LIN {X 0,Y 453.456,Z 225.499,A -85,B 0,C 180,E1 -8413.244,E2 -8413.244} C_VEL
LIN {X 0,Y 453.465,Z 225.498,A -85,B 0,C 180,E1 -8415.778,E2 -8415.778} C_VEL
LIN {X 0,Y 453.48,Z 225.494,A -85,B 0,C 180,E1 -8418.209,E2 -8418.209} C_VEL
LIN {X 0,Y 453.488,Z 225.488,A -85,B 0,C 180,E1 -8420.794,E2 -8420.794} C_VEL
LIN {X 0,Y 453.455,Z 225.496,A -85,B 0,C 180,E1 -8423.917,E2 -8423.917} C_VEL
LIN {X 0,Y 453.475,Z 225.49,A -85,B 0,C 180,E1 -8427.15,E2 -8427.15} C_VEL
LIN {X 0,Y 453.475,Z 225.494,A -85,B 0,C 180,E1 -8430.268,E2 -8430.268} C_VEL
LIN {X 0,Y 453.504,Z 225.483,A -85,B 0,C 180,E1 -8433.293,E2 -8433.293} C_VEL
LIN {X 0,Y 453.502,Z 225.49,A -85,B 0,C 180,E1 -8436.238,E2 -8436.238} C_VEL
LIN {X 0,Y 453.483,Z 225.493,A -85,B 0,C 180,E1 -8439.117,E2 -8439.117} C_VEL
LIN {X 0,Y 453.503,Z 225.478,A -85,B 0,C 180,E1 -8441.944,E2 -8441.944} C_VEL
LIN {X 0,Y 453.54,Z 225.486,A -85,B 0,C 180,E1 -8444.726,E2 -8444.726} C_VEL
LIN {X 0,Y 453.559,Z 225.479,A -85,B 0,C 180,E1 -8448.378,E2 -8448.378} C_VEL
LIN {X 0,Y 453.585,Z 225.469,A -85,B 0,C 180,E1 -8451.086,E2 -8451.086} C_VEL
LIN {X 0,Y 453.653,Z 225.471,A -85,B 0,C 180,E1 -8453.774,E2 -8453.774} C_VEL
LIN {X 0,Y 453.744,Z 225.458,A -85,B 0,C 180,E1 -8457.336,E2 -8457.336} C_VEL
LIN {X 0,Y 453.822,Z 225.434,A -85,B 0,C 180,E1 -8460,E2 -8460} C_VEL
LIN {X 0,Y 453.763,Z 225.456,A -85,B 0,C 180,E1 -8462.663,E2 -8462.663} C_VEL
LIN {X 0,Y 453.669,Z 225.472,A -85,B 0,C 180,E1 -8466.225,E2 -8466.225} C_VEL
LIN {X 0,Y 453.591,Z 225.467,A -85,B 0,C 180,E1 -8468.913,E2 -8468.913} C_VEL
LIN {X 0,Y 453.562,Z 225.483,A -85,B 0,C 180,E1 -8472.528,E2 -8472.528} C_VEL
LIN {X 0,Y 453.543,Z 225.49,A -85,B 0,C 180,E1 -8476.195,E2 -8476.195} C_VEL
LIN {X 0,Y 453.518,Z 225.475,A -85,B 0,C 180,E1 -8479.04,E2 -8479.04} C_VEL
LIN {X 0,Y 453.474,Z 225.493,A -85,B 0,C 180,E1 -8481.836,E2 -8481.836} C_VEL
LIN {X 0,Y 453.498,Z 225.491,A -85,B 0,C 180,E1 -8484.735,E2 -8484.735} C_VEL
LIN {X 0,Y 453.529,Z 225.478,A -85,B 0,C 180,E1 -8487.959,E2 -8487.959} C_VEL
LIN {X 0,Y 453.463,Z 225.498,A -85,B 0,C 180,E1 -8491.525,E2 -8491.525} C_VEL
LIN {X 0,Y 453.485,Z 225.487,A -85,B 0,C 180,E1 -8494.777,E2 -8494.777} C_VEL
LIN {X 0,Y 453.47,Z 225.499,A -85,B 0,C 180,E1 -8498.31,E2 -8498.31} C_VEL
LIN {X 0,Y 453.491,Z 225.487,A -85,B 0,C 180,E1 -8500.609,E2 -8500.609} C_VEL
LIN {X 0,Y 453.478,Z 225.495,A -85,B 0,C 180,E1 -8503.247,E2 -8503.247} C_VEL
LIN {X 0,Y 453.462,Z 225.49,A -85,B 0,C 180,E1 -8505.779,E2 -8505.779} C_VEL
LIN {X 0,Y 453.512,Z 225.476,A -85,B 0,C 180,E1 -8509.405,E2 -8509.405} C_VEL
LIN {X 0,Y 453.473,Z 225.498,A -85,B 0,C 180,E1 -8512.223,E2 -8512.223} C_VEL
LIN {X 0,Y 453.485,Z 225.482,A -85,B 0,C 180,E1 -8515.222,E2 -8515.222} C_VEL
LIN {X 0,Y 453.463,Z 225.497,A -85,B 0,C 180,E1 -8518.474,E2 -8518.474} C_VEL
LIN {X 0,Y 453.534,Z 225.491,A -85,B 0,C 180,E1 -8522.039,E2 -8522.039} C_VEL
LIN {X 0,Y 453.51,Z 225.496,A -85,B 0,C 180,E1 -8525.265,E2 -8525.265} C_VEL
LIN {X 0,Y 453.476,Z 225.497,A -85,B 0,C 180,E1 -8528.415,E2 -8528.415} C_VEL
LIN {X 0,Y 453.519,Z 225.495,A -85,B 0,C 180,E1 -8531.009,E2 -8531.009} C_VEL
LIN {X 0,Y 453.565,Z 225.488,A -85,B 0,C 180,E1 -8533.88,E2 -8533.88} C_VEL
LIN {X 0,Y 453.56,Z 225.49,A -85,B 0,C 180,E1 -8537.471,E2 -8537.471} C_VEL
LIN {X 0,Y 453.589,Z 225.487,A -85,B 0,C 180,E1 -8541.087,E2 -8541.087} C_VEL
LIN {X 0,Y 453.634,Z 225.48,A -85,B 0,C 180,E1 -8543.088,E2 -8543.088} C_VEL
LIN {X 0,Y 452.949,Z 225.565,A -85,B 0,C 180,E1 -8543.829,E2 -8543.829} C_VEL
LIN {X 0,Y 450,Z 225.934,A -85,B 0,C 180,E1 -8545.03,E2 -8545.03} C_VEL
LIN {X 0,Y 447.577,Z 226.234,A -85,B 0,C 180,E1 -8546,E2 -8546} C_VEL
LIN {X 0,Y 446.64,Z 226.352,A -85,B 0,C 180,E1 -8546.75,E2 -8546.75} C_VEL
LIN {X 0,Y 446.62,Z 226.353,A -85,B 0,C 180,E1 -8547.004,E2 -8547.004} C_VEL
LIN {X 0,Y 446.791,Z 226.332,A -85,B 0,C 180,E1 -8550,E2 -8550} C_VEL
LIN {X 0,Y 446.706,Z 226.344,A -85,B 0,C 180,E1 -8552.705,E2 -8552.705} C_VEL
LIN {X 0,Y 446.645,Z 226.351,A -85,B 0,C 180,E1 -8556.324,E2 -8556.324} C_VEL
LIN {X 0,Y 446.535,Z 226.365,A -85,B 0,C 180,E1 -8559.055,E2 -8559.055} C_VEL
LIN {X 0,Y 446.518,Z 226.368,A -85,B 0,C 180,E1 -8562.73,E2 -8562.73} C_VEL
LIN {X 0,Y 446.492,Z 226.37,A -85,B 0,C 180,E1 -8566.228,E2 -8566.228} C_VEL
LIN {X 0,Y 446.466,Z 226.371,A -85,B 0,C 180,E1 -8569.303,E2 -8569.303} C_VEL
LIN {X 0,Y 446.414,Z 226.38,A -85,B 0,C 180,E1 -8572.2,E2 -8572.2} C_VEL
LIN {X 0,Y 446.453,Z 226.372,A -85,B 0,C 180,E1 -8575.152,E2 -8575.152} C_VEL
LIN {X 0,Y 446.481,Z 226.365,A -85,B 0,C 180,E1 -8578.179,E2 -8578.179} C_VEL
LIN {X 0,Y 446.416,Z 226.377,A -85,B 0,C 180,E1 -8581.775,E2 -8581.775} C_VEL
LIN {X 0,Y 446.426,Z 226.36,A -85,B 0,C 180,E1 -8584.523,E2 -8584.523} C_VEL
LIN {X 0,Y 446.432,Z 226.378,A -85,B 0,C 180,E1 -8588.083,E2 -8588.083} C_VEL
LIN {X 0,Y 446.439,Z 226.355,A -85,B 0,C 180,E1 -8590.92,E2 -8590.92} C_VEL
LIN {X 0,Y 446.398,Z 226.364,A -85,B 0,C 180,E1 -8593.846,E2 -8593.846} C_VEL
LIN {X 0,Y 446.443,Z 226.374,A -85,B 0,C 180,E1 -8596.397,E2 -8596.397} C_VEL
LIN {X 0,Y 446.464,Z 226.364,A -85,B 0,C 180,E1 -8599.805,E2 -8599.805} C_VEL
LIN {X 0,Y 446.428,Z 226.378,A -85,B 0,C 180,E1 -8602.124,E2 -8602.124} C_VEL
LIN {X 0,Y 446.427,Z 226.366,A -85,B 0,C 180,E1 -8605.477,E2 -8605.477} C_VEL
LIN {X 0,Y 446.413,Z 226.375,A -85,B 0,C 180,E1 -8608.7,E2 -8608.7} C_VEL
LIN {X 0,Y 446.482,Z 226.358,A -85,B 0,C 180,E1 -8611.822,E2 -8611.822} C_VEL
LIN {X 0,Y 446.441,Z 226.368,A -85,B 0,C 180,E1 -8614.847,E2 -8614.847} C_VEL
LIN {X 0,Y 446.446,Z 226.367,A -85,B 0,C 180,E1 -8618.246,E2 -8618.246} C_VEL
LIN {X 0,Y 446.455,Z 226.359,A -85,B 0,C 180,E1 -8621.65,E2 -8621.65} C_VEL
LIN {X 0,Y 446.507,Z 226.362,A -85,B 0,C 180,E1 -8624.48,E2 -8624.48} C_VEL
LIN {X 0,Y 446.516,Z 226.353,A -85,B 0,C 180,E1 -8628.194,E2 -8628.194} C_VEL
LIN {X 0,Y 446.599,Z 226.347,A -85,B 0,C 180,E1 -8631.858,E2 -8631.858} C_VEL
LIN {X 0,Y 446.641,Z 226.346,A -85,B 0,C 180,E1 -8634.583,E2 -8634.583} C_VEL
LIN {X 0,Y 446.707,Z 226.335,A -85,B 0,C 180,E1 -8637.295,E2 -8637.295} C_VEL
LIN {X 0,Y 446.792,Z 226.309,A -85,B 0,C 180,E1 -8640,E2 -8640} C_VEL
LIN {X 0,Y 446.691,Z 226.336,A -85,B 0,C 180,E1 -8642.706,E2 -8642.706} C_VEL
LIN {X 0,Y 446.621,Z 226.347,A -85,B 0,C 180,E1 -8646.325,E2 -8646.325} C_VEL
LIN {X 0,Y 446.52,Z 226.343,A -85,B 0,C 180,E1 -8649.971,E2 -8649.971} C_VEL
LIN {X 0,Y 446.521,Z 226.36,A -85,B 0,C 180,E1 -8652.73,E2 -8652.73} C_VEL
LIN {X 0,Y 446.496,Z 226.361,A -85,B 0,C 180,E1 -8656.228,E2 -8656.228} C_VEL
LIN {X 0,Y 446.468,Z 226.358,A -85,B 0,C 180,E1 -8659.304,E2 -8659.304} C_VEL
LIN {X 0,Y 446.418,Z 226.373,A -85,B 0,C 180,E1 -8662.2,E2 -8662.2} C_VEL
LIN {X 0,Y 446.45,Z 226.364,A -85,B 0,C 180,E1 -8665.153,E2 -8665.153} C_VEL
LIN {X 0,Y 446.485,Z 226.358,A -85,B 0,C 180,E1 -8668.179,E2 -8668.179} C_VEL
LIN {X 0,Y 446.415,Z 226.374,A -85,B 0,C 180,E1 -8671.301,E2 -8671.301} C_VEL
LIN {X 0,Y 446.423,Z 226.368,A -85,B 0,C 180,E1 -8674.524,E2 -8674.524} C_VEL
LIN {X 0,Y 446.414,Z 226.378,A -85,B 0,C 180,E1 -8678.079,E2 -8678.079} C_VEL
LIN {X 0,Y 446.428,Z 226.373,A -85,B 0,C 180,E1 -8680.918,E2 -8680.918} C_VEL
LIN {X 0,Y 446.401,Z 226.377,A -85,B 0,C 180,E1 -8683.846,E2 -8683.846} C_VEL
LIN {X 0,Y 446.4,Z 226.382,A -85,B 0,C 180,E1 -8686.404,E2 -8686.404} C_VEL
LIN {X 0,Y 446.428,Z 226.361,A -85,B 0,C 180,E1 -8689.083,E2 -8689.083} C_VEL
LIN {X 0,Y 446.418,Z 226.377,A -85,B 0,C 180,E1 -8691.921,E2 -8691.921} C_VEL
LIN {X 0,Y 446.431,Z 226.372,A -85,B 0,C 180,E1 -8695.477,E2 -8695.477} C_VEL
LIN {X 0,Y 446.418,Z 226.38,A -85,B 0,C 180,E1 -8698.7,E2 -8698.7} C_VEL
LIN {X 0,Y 446.523,Z 226.546,A -85,B 0,C 180,E1 -8701.824,E2 -8701.824} C_VEL
LIN {X 0,Y 448.351,Z 236.652,A -85,B 0,C 180,E1 -8704.465,E2 -8704.465} C_VEL
LIN {X 0,Y 448.414,Z 241.452,A -85,B 0,C 180,E1 -8705.652,E2 -8705.652} C_VEL
LIN {X 0,Y 447.64,Z 256.177,A -85,B 0,C 180,E1 -8709.073,E2 -8709.073} C_VEL
LIN {X 0,Y 446.976,Z 268.254,A -85,B 0,C 180,E1 -8711.909,E2 -8711.909} C_VEL
LIN {X 0,Y 446.96,Z 269.57,A -85,B 0,C 180,E1 -8712.145,E2 -8712.145} C_VEL
LIN {X 0,Y 450.754,Z 291.489,A -85,B 0,C 180,E1 -8712.682,E2 -8712.682} C_VEL
LIN {X 0,Y 450.084,Z 374.211,A -85,B 0,C 180,E1 -8714.025,E2 -8714.025} C_VEL
LIN {X 0,Y 449.785,Z 384.982,A -85,B 0,C 180,E1 -8714.305,E2 -8714.305} C_VEL
LIN {X 0,Y 449.46,Z 394.085,A -85,B 0,C 180,E1 -8714.642,E2 -8714.642} C_VEL
LIN {X 0,Y 449.017,Z 403.44,A -85,B 0,C 180,E1 -8715.091,E2 -8715.091} C_VEL
LIN {X 0,Y 448.546,Z 413.584,A -85,B 0,C 180,E1 -8715.713,E2 -8715.713} C_VEL
LIN {X 0,Y 448.03,Z 422.582,A -85,B 0,C 180,E1 -8716.391,E2 -8716.391} C_VEL
LIN {X 0,Y 447.593,Z 431.188,A -85,B 0,C 180,E1 -8717.173,E2 -8717.173} C_VEL
LIN {X 0,Y 447.167,Z 438.71,A -85,B 0,C 180,E1 -8717.98,E2 -8717.98} C_VEL
LIN {X 0,Y 446.682,Z 445.929,A -85,B 0,C 180,E1 -8718.887,E2 -8718.887} C_VEL
LIN {X 0,Y 446.366,Z 452.133,A -85,B 0,C 180,E1 -8719.797,E2 -8719.797} C_VEL
LIN {X 0,Y 446.002,Z 458.67,A -85,B 0,C 180,E1 -8720.934,E2 -8720.934} C_VEL
LIN {X 0,Y 445.788,Z 463.171,A -85,B 0,C 180,E1 -8721.843,E2 -8721.843} C_VEL
LIN {X 0,Y 445.573,Z 468.664,A -85,B 0,C 180,E1 -8723.207,E2 -8723.207} C_VEL
LIN {X 0,Y 445.476,Z 472.985,A -85,B 0,C 180,E1 -8724.568,E2 -8724.568} C_VEL
LIN {X 0,Y 445.413,Z 475.35,A -85,B 0,C 180,E1 -8725.475,E2 -8725.475} C_VEL
LIN {X 0,Y 445.433,Z 478.533,A -85,B 0,C 180,E1 -8727.287,E2 -8727.287} C_VEL
LIN {X 0,Y 445.356,Z 479.588,A -85,B 0,C 180,E1 -8728.191,E2 -8728.191} C_VEL
LIN {X 0,Y 445.339,Z 480.175,A -85,B 0,C 180,E1 -8729.096,E2 -8729.096} C_VEL
LIN {X 0,Y 445.339,Z 480.175,A -85,B 0,C 180,E1 -8730.904,E2 -8730.904} C_VEL
LIN {X 0,Y 445.356,Z 479.588,A -85,B 0,C 180,E1 -8731.809,E2 -8731.809} C_VEL
LIN {X 0,Y 445.433,Z 478.533,A -85,B 0,C 180,E1 -8732.713,E2 -8732.713} C_VEL
LIN {X 0,Y 445.413,Z 475.35,A -85,B 0,C 180,E1 -8734.525,E2 -8734.525} C_VEL
LIN {X 0,Y 445.469,Z 471.235,A -85,B 0,C 180,E1 -8736.042,E2 -8736.042} C_VEL
LIN {X 0,Y 445.601,Z 467.001,A -85,B 0,C 180,E1 -8737.249,E2 -8737.249} C_VEL
LIN {X 0,Y 445.892,Z 460.981,A -85,B 0,C 180,E1 -8738.612,E2 -8738.612} C_VEL
LIN {X 0,Y 446.208,Z 454.885,A -85,B 0,C 180,E1 -8739.748,E2 -8739.748} C_VEL
LIN {X 0,Y 446.49,Z 449.183,A -85,B 0,C 180,E1 -8740.658,E2 -8740.658} C_VEL
LIN {X 0,Y 447.026,Z 440.629,A -85,B 0,C 180,E1 -8741.793,E2 -8741.793} C_VEL
LIN {X 0,Y 447.504,Z 432.448,A -85,B 0,C 180,E1 -8742.701,E2 -8742.701} C_VEL
LIN {X 0,Y 447.964,Z 424.011,A -85,B 0,C 180,E1 -8743.489,E2 -8743.489} C_VEL
LIN {X 0,Y 448.424,Z 415.215,A -85,B 0,C 180,E1 -8744.175,E2 -8744.175} C_VEL
LIN {X 0,Y 448.928,Z 405.455,A -85,B 0,C 180,E1 -8744.796,E2 -8744.796} C_VEL
LIN {X 0,Y 449.374,Z 395.371,A -85,B 0,C 180,E1 -8745.303,E2 -8745.303} C_VEL
LIN {X 0,Y 449.794,Z 385.857,A -85,B 0,C 180,E1 -8745.665,E2 -8745.665} C_VEL
LIN {X 0,Y 450.066,Z 376.876,A -85,B 0,C 180,E1 -8745.917,E2 -8745.917} C_VEL
LIN {X 0,Y 450.302,Z 351.751,A -85,B 0,C 180,E1 -8746.353,E2 -8746.353} C_VEL
LIN {X 0,Y 450.679,Z 291.103,A -85,B 0,C 180,E1 -8747.327,E2 -8747.327} C_VEL
LIN {X 0,Y 446.993,Z 269.773,A -85,B 0,C 180,E1 -8747.84,E2 -8747.84} C_VEL
LIN {X 0,Y 446.946,Z 268.723,A -85,B 0,C 180,E1 -8747.977,E2 -8747.977} C_VEL
LIN {X 0,Y 447.701,Z 255.359,A -85,B 0,C 180,E1 -8751.165,E2 -8751.165} C_VEL
LIN {X 0,Y 448.56,Z 240.272,A -85,B 0,C 180,E1 -8754.667,E2 -8754.667} C_VEL
LIN {X 0,Y 448.185,Z 235.634,A -85,B 0,C 180,E1 -8755.795,E2 -8755.795} C_VEL
LIN {X 0,Y 446.512,Z 226.436,A -85,B 0,C 180,E1 -8758.228,E2 -8758.228} C_VEL
LIN {X 0,Y 446.422,Z 226.375,A -85,B 0,C 180,E1 -8761.775,E2 -8761.775} C_VEL
LIN {X 0,Y 446.431,Z 226.373,A -85,B 0,C 180,E1 -8764.523,E2 -8764.523} C_VEL
LIN {X 0,Y 446.418,Z 226.378,A -85,B 0,C 180,E1 -8768.079,E2 -8768.079} C_VEL
LIN {X 0,Y 446.428,Z 226.36,A -85,B 0,C 180,E1 -8770.917,E2 -8770.917} C_VEL
LIN {X 0,Y 446.402,Z 226.381,A -85,B 0,C 180,E1 -8773.846,E2 -8773.846} C_VEL
LIN {X 0,Y 446.399,Z 226.376,A -85,B 0,C 180,E1 -8776.403,E2 -8776.403} C_VEL
LIN {X 0,Y 446.428,Z 226.373,A -85,B 0,C 180,E1 -8779.082,E2 -8779.082} C_VEL
LIN {X 0,Y 446.408,Z 226.377,A -85,B 0,C 180,E1 -8782.121,E2 -8782.121} C_VEL
LIN {X 0,Y 446.423,Z 226.368,A -85,B 0,C 180,E1 -8785.476,E2 -8785.476} C_VEL
LIN {X 0,Y 446.415,Z 226.374,A -85,B 0,C 180,E1 -8788.699,E2 -8788.699} C_VEL
LIN {X 0,Y 446.485,Z 226.358,A -85,B 0,C 180,E1 -8791.821,E2 -8791.821} C_VEL
LIN {X 0,Y 446.45,Z 226.364,A -85,B 0,C 180,E1 -8794.847,E2 -8794.847} C_VEL
LIN {X 0,Y 446.448,Z 226.367,A -85,B 0,C 180,E1 -8798.245,E2 -8798.245} C_VEL
LIN {X 0,Y 446.452,Z 226.357,A -85,B 0,C 180,E1 -8801.648,E2 -8801.648} C_VEL
LIN {X 0,Y 446.508,Z 226.359,A -85,B 0,C 180,E1 -8804.479,E2 -8804.479} C_VEL
LIN {X 0,Y 446.517,Z 226.355,A -85,B 0,C 180,E1 -8808.193,E2 -8808.193} C_VEL
LIN {X 0,Y 446.532,Z 226.345,A -85,B 0,C 180,E1 -8810.944,E2 -8810.944} C_VEL
LIN {X 0,Y 446.621,Z 226.347,A -85,B 0,C 180,E1 -8813.675,E2 -8813.675} C_VEL
LIN {X 0,Y 446.691,Z 226.336,A -85,B 0,C 180,E1 -8817.294,E2 -8817.294} C_VEL
LIN {X 0,Y 446.792,Z 226.309,A -85,B 0,C 180,E1 -8820,E2 -8820} C_VEL
LIN {X 0,Y 446.707,Z 226.335,A -85,B 0,C 180,E1 -8822.705,E2 -8822.705} C_VEL
LIN {X 0,Y 446.638,Z 226.349,A -85,B 0,C 180,E1 -8826.323,E2 -8826.323} C_VEL
LIN {X 0,Y 446.537,Z 226.343,A -85,B 0,C 180,E1 -8829.055,E2 -8829.055} C_VEL
LIN {X 0,Y 446.52,Z 226.363,A -85,B 0,C 180,E1 -8832.729,E2 -8832.729} C_VEL
LIN {X 0,Y 446.494,Z 226.368,A -85,B 0,C 180,E1 -8836.227,E2 -8836.227} C_VEL
LIN {X 0,Y 446.467,Z 226.352,A -85,B 0,C 180,E1 -8839.303,E2 -8839.303} C_VEL
LIN {X 0,Y 446.415,Z 226.376,A -85,B 0,C 180,E1 -8842.199,E2 -8842.199} C_VEL
LIN {X 0,Y 446.441,Z 226.367,A -85,B 0,C 180,E1 -8845.153,E2 -8845.153} C_VEL
LIN {X 0,Y 446.482,Z 226.358,A -85,B 0,C 180,E1 -8848.178,E2 -8848.178} C_VEL
LIN {X 0,Y 446.416,Z 226.378,A -85,B 0,C 180,E1 -8851.775,E2 -8851.775} C_VEL
LIN {X 0,Y 446.427,Z 226.366,A -85,B 0,C 180,E1 -8854.523,E2 -8854.523} C_VEL
LIN {X 0,Y 446.427,Z 226.379,A -85,B 0,C 180,E1 -8858.081,E2 -8858.081} C_VEL
LIN {X 0,Y 446.425,Z 226.366,A -85,B 0,C 180,E1 -8860.918,E2 -8860.918} C_VEL
LIN {X 0,Y 446.442,Z 226.377,A -85,B 0,C 180,E1 -8863.84,E2 -8863.84} C_VEL
LIN {X 0,Y 446.395,Z 226.362,A -85,B 0,C 180,E1 -8866.403,E2 -8866.403} C_VEL
LIN {X 0,Y 446.464,Z 226.359,A -85,B 0,C 180,E1 -8869.805,E2 -8869.805} C_VEL
LIN {X 0,Y 446.428,Z 226.376,A -85,B 0,C 180,E1 -8872.123,E2 -8872.123} C_VEL
LIN {X 0,Y 446.426,Z 226.36,A -85,B 0,C 180,E1 -8875.477,E2 -8875.477} C_VEL
LIN {X 0,Y 446.413,Z 226.376,A -85,B 0,C 180,E1 -8878.7,E2 -8878.7} C_VEL
LIN {X 0,Y 446.481,Z 226.366,A -85,B 0,C 180,E1 -8881.821,E2 -8881.821} C_VEL
LIN {X 0,Y 446.453,Z 226.372,A -85,B 0,C 180,E1 -8884.848,E2 -8884.848} C_VEL
LIN {X 0,Y 446.444,Z 226.373,A -85,B 0,C 180,E1 -8888.245,E2 -8888.245} C_VEL
LIN {X 0,Y 446.454,Z 226.375,A -85,B 0,C 180,E1 -8891.649,E2 -8891.649} C_VEL
LIN {X 0,Y 446.505,Z 226.367,A -85,B 0,C 180,E1 -8894.48,E2 -8894.48} C_VEL
LIN {X 0,Y 446.514,Z 226.366,A -85,B 0,C 180,E1 -8898.193,E2 -8898.193} C_VEL
LIN {X 0,Y 446.597,Z 226.357,A -85,B 0,C 180,E1 -8901.858,E2 -8901.858} C_VEL
LIN {X 0,Y 446.644,Z 226.351,A -85,B 0,C 180,E1 -8904.583,E2 -8904.583} C_VEL
LIN {X 0,Y 446.62,Z 226.353,A -85,B 0,C 180,E1 -8907.004,E2 -8907.004} C_VEL
LIN {X 0,Y 446.102,Z 226.421,A -85,B 0,C 180,E1 -8907.757,E2 -8907.757} C_VEL
LIN {X 0,Y 443.287,Z 226.776,A -85,B 0,C 180,E1 -8908.98,E2 -8908.98} C_VEL
LIN {X 0,Y 440.802,Z 227.085,A -85,B 0,C 180,E1 -8909.966,E2 -8909.966} C_VEL
LIN {X 0,Y 439.713,Z 227.217,A -85,B 0,C 180,E1 -8910.73,E2 -8910.73} C_VEL
LIN {X 0,Y 439.619,Z 227.226,A -85,B 0,C 180,E1 -8910.989,E2 -8910.989} C_VEL
LIN {X 0,Y 439.653,Z 227.222,A -85,B 0,C 180,E1 -8912.749,E2 -8912.749} C_VEL
LIN {X 0,Y 439.616,Z 227.227,A -85,B 0,C 180,E1 -8916.425,E2 -8916.425} C_VEL
LIN {X 0,Y 439.497,Z 227.242,A -85,B 0,C 180,E1 -8919.202,E2 -8919.202} C_VEL
LIN {X 0,Y 439.462,Z 227.246,A -85,B 0,C 180,E1 -8922.938,E2 -8922.938} C_VEL
LIN {X 0,Y 439.444,Z 227.249,A -85,B 0,C 180,E1 -8926.349,E2 -8926.349} C_VEL
LIN {X 0,Y 439.399,Z 227.251,A -85,B 0,C 180,E1 -8929.626,E2 -8929.626} C_VEL
LIN {X 0,Y 439.361,Z 227.26,A -85,B 0,C 180,E1 -8932.576,E2 -8932.576} C_VEL
LIN {X 0,Y 439.401,Z 227.25,A -85,B 0,C 180,E1 -8935.585,E2 -8935.585} C_VEL
LIN {X 0,Y 439.414,Z 227.237,A -85,B 0,C 180,E1 -8938.674,E2 -8938.674} C_VEL
LIN {X 0,Y 439.367,Z 227.257,A -85,B 0,C 180,E1 -8942.031,E2 -8942.031} C_VEL
LIN {X 0,Y 439.392,Z 227.237,A -85,B 0,C 180,E1 -8945.341,E2 -8945.341} C_VEL
LIN {X 0,Y 439.392,Z 227.251,A -85,B 0,C 180,E1 -8948.594,E2 -8948.594} C_VEL
LIN {X 0,Y 439.394,Z 227.23,A -85,B 0,C 180,E1 -8951.259,E2 -8951.259} C_VEL
LIN {X 0,Y 439.399,Z 227.246,A -85,B 0,C 180,E1 -8954.729,E2 -8954.729} C_VEL
LIN {X 0,Y 439.406,Z 227.252,A -85,B 0,C 180,E1 -8957.798,E2 -8957.798} C_VEL
LIN {X 0,Y 439.446,Z 227.243,A -85,B 0,C 180,E1 -8960.23,E2 -8960.23} C_VEL
LIN {X 0,Y 439.374,Z 227.255,A -85,B 0,C 180,E1 -8963.714,E2 -8963.714} C_VEL
LIN {X 0,Y 439.369,Z 227.248,A -85,B 0,C 180,E1 -8967.054,E2 -8967.054} C_VEL
LIN {X 0,Y 439.379,Z 227.249,A -85,B 0,C 180,E1 -8970.275,E2 -8970.275} C_VEL
LIN {X 0,Y 439.425,Z 227.233,A -85,B 0,C 180,E1 -8973.397,E2 -8973.397} C_VEL
LIN {X 0,Y 439.381,Z 227.251,A -85,B 0,C 180,E1 -8976.43,E2 -8976.43} C_VEL
LIN {X 0,Y 439.387,Z 227.245,A -85,B 0,C 180,E1 -8979.398,E2 -8979.398} C_VEL
LIN {X 0,Y 439.429,Z 227.237,A -85,B 0,C 180,E1 -8982.31,E2 -8982.31} C_VEL
LIN {X 0,Y 439.447,Z 227.245,A -85,B 0,C 180,E1 -8985.175,E2 -8985.175} C_VEL
LIN {X 0,Y 439.482,Z 227.23,A -85,B 0,C 180,E1 -8988.002,E2 -8988.002} C_VEL
LIN {X 0,Y 439.547,Z 227.226,A -85,B 0,C 180,E1 -8991.727,E2 -8991.727} C_VEL
LIN {X 0,Y 439.617,Z 227.221,A -85,B 0,C 180,E1 -8994.496,E2 -8994.496} C_VEL
LIN {X 0,Y 439.634,Z 227.208,A -85,B 0,C 180,E1 -8998.168,E2 -8998.168} C_VEL
LIN {X 0,Y 439.762,Z 227.184,A -85,B 0,C 180,E1 -9000.001,E2 -9000.001} C_VEL
LIN {X 0,Y 439.64,Z 227.215,A -85,B 0,C 180,E1 -9002.749,E2 -9002.749} C_VEL
LIN {X 0,Y 439.592,Z 227.223,A -85,B 0,C 180,E1 -9006.426,E2 -9006.426} C_VEL
LIN {X 0,Y 439.495,Z 227.22,A -85,B 0,C 180,E1 -9009.202,E2 -9009.202} C_VEL
LIN {X 0,Y 439.465,Z 227.241,A -85,B 0,C 180,E1 -9012.938,E2 -9012.938} C_VEL
LIN {X 0,Y 439.446,Z 227.24,A -85,B 0,C 180,E1 -9016.349,E2 -9016.349} C_VEL
LIN {X 0,Y 439.402,Z 227.237,A -85,B 0,C 180,E1 -9019.627,E2 -9019.627} C_VEL
LIN {X 0,Y 439.365,Z 227.255,A -85,B 0,C 180,E1 -9022.576,E2 -9022.576} C_VEL
LIN {X 0,Y 439.401,Z 227.239,A -85,B 0,C 180,E1 -9025.586,E2 -9025.586} C_VEL
LIN {X 0,Y 439.418,Z 227.244,A -85,B 0,C 180,E1 -9028.674,E2 -9028.674} C_VEL
LIN {X 0,Y 439.366,Z 227.253,A -85,B 0,C 180,E1 -9032.03,E2 -9032.03} C_VEL
LIN {X 0,Y 439.393,Z 227.245,A -85,B 0,C 180,E1 -9035.34,E2 -9035.34} C_VEL
LIN {X 0,Y 439.376,Z 227.251,A -85,B 0,C 180,E1 -9038.596,E2 -9038.596} C_VEL
LIN {X 0,Y 439.389,Z 227.248,A -85,B 0,C 180,E1 -9041.257,E2 -9041.257} C_VEL
LIN {X 0,Y 439.401,Z 227.249,A -85,B 0,C 180,E1 -9044.73,E2 -9044.73} C_VEL
LIN {X 0,Y 439.397,Z 227.251,A -85,B 0,C 180,E1 -9047.796,E2 -9047.796} C_VEL
LIN {X 0,Y 439.432,Z 227.235,A -85,B 0,C 180,E1 -9050.228,E2 -9050.228} C_VEL
LIN {X 0,Y 439.376,Z 227.25,A -85,B 0,C 180,E1 -9053.713,E2 -9053.713} C_VEL
LIN {X 0,Y 439.375,Z 227.251,A -85,B 0,C 180,E1 -9057.054,E2 -9057.054} C_VEL
LIN {X 0,Y 439.38,Z 227.251,A -85,B 0,C 180,E1 -9060.274,E2 -9060.274} C_VEL
LIN {X 0,Y 439.464,Z 227.427,A -85,B 0,C 180,E1 -9061.592,E2 -9061.592} C_VEL
LIN {X 0,Y 441.164,Z 236.51,A -85,B 0,C 180,E1 -9064.018,E2 -9064.018} C_VEL
LIN {X 0,Y 441.543,Z 240.8,A -85,B 0,C 180,E1 -9065.131,E2 -9065.131} C_VEL
LIN {X 0,Y 440.741,Z 254.975,A -85,B 0,C 180,E1 -9068.484,E2 -9068.484} C_VEL
LIN {X 0,Y 440.058,Z 267.11,A -85,B 0,C 180,E1 -9071.373,E2 -9071.373} C_VEL
LIN {X 0,Y 439.98,Z 269.101,A -85,B 0,C 180,E1 -9071.822,E2 -9071.822} C_VEL
LIN {X 0,Y 440.538,Z 272.624,A -85,B 0,C 180,E1 -9071.956,E2 -9071.956} C_VEL
LIN {X 0,Y 443.97,Z 293,A -85,B 0,C 180,E1 -9072.437,E2 -9072.437} C_VEL
LIN {X 0,Y 443.27,Z 374.019,A -85,B 0,C 180,E1 -9073.773,E2 -9073.773} C_VEL
LIN {X 0,Y 442.995,Z 383.915,A -85,B 0,C 180,E1 -9074.029,E2 -9074.029} C_VEL
LIN {X 0,Y 442.624,Z 393.892,A -85,B 0,C 180,E1 -9074.399,E2 -9074.399} C_VEL
LIN {X 0,Y 442.165,Z 403.248,A -85,B 0,C 180,E1 -9074.855,E2 -9074.855} C_VEL
LIN {X 0,Y 441.652,Z 413.391,A -85,B 0,C 180,E1 -9075.485,E2 -9075.485} C_VEL
LIN {X 0,Y 441.113,Z 422.388,A -85,B 0,C 180,E1 -9076.173,E2 -9076.173} C_VEL
LIN {X 0,Y 440.676,Z 430.523,A -85,B 0,C 180,E1 -9076.92,E2 -9076.92} C_VEL
LIN {X 0,Y 440.198,Z 438.517,A -85,B 0,C 180,E1 -9077.787,E2 -9077.787} C_VEL
LIN {X 0,Y 439.699,Z 445.736,A -85,B 0,C 180,E1 -9078.709,E2 -9078.709} C_VEL
LIN {X 0,Y 439.343,Z 451.939,A -85,B 0,C 180,E1 -9079.633,E2 -9079.633} C_VEL
LIN {X 0,Y 438.974,Z 458.477,A -85,B 0,C 180,E1 -9080.787,E2 -9080.787} C_VEL
LIN {X 0,Y 438.741,Z 462.978,A -85,B 0,C 180,E1 -9081.711,E2 -9081.711} C_VEL
LIN {X 0,Y 438.501,Z 468.469,A -85,B 0,C 180,E1 -9083.096,E2 -9083.096} C_VEL
LIN {X 0,Y 438.374,Z 472.792,A -85,B 0,C 180,E1 -9084.48,E2 -9084.48} C_VEL
LIN {X 0,Y 438.342,Z 475.157,A -85,B 0,C 180,E1 -9085.402,E2 -9085.402} C_VEL
LIN {X 0,Y 438.341,Z 478.341,A -85,B 0,C 180,E1 -9087.243,E2 -9087.243} C_VEL
LIN {X 0,Y 438.279,Z 479.396,A -85,B 0,C 180,E1 -9088.162,E2 -9088.162} C_VEL
LIN {X 0,Y 438.253,Z 479.983,A -85,B 0,C 180,E1 -9089.081,E2 -9089.081} C_VEL
LIN {X 0,Y 438.253,Z 479.983,A -85,B 0,C 180,E1 -9090.919,E2 -9090.919} C_VEL
LIN {X 0,Y 438.279,Z 479.396,A -85,B 0,C 180,E1 -9091.838,E2 -9091.838} C_VEL
LIN {X 0,Y 438.341,Z 478.341,A -85,B 0,C 180,E1 -9092.757,E2 -9092.757} C_VEL
LIN {X 0,Y 438.342,Z 475.157,A -85,B 0,C 180,E1 -9094.598,E2 -9094.598} C_VEL
LIN {X 0,Y 438.423,Z 470.356,A -85,B 0,C 180,E1 -9096.343,E2 -9096.343} C_VEL
LIN {X 0,Y 438.634,Z 464.893,A -85,B 0,C 180,E1 -9097.827,E2 -9097.827} C_VEL
LIN {X 0,Y 438.895,Z 459.632,A -85,B 0,C 180,E1 -9098.982,E2 -9098.982} C_VEL
LIN {X 0,Y 439.262,Z 453.315,A -85,B 0,C 180,E1 -9100.137,E2 -9100.137} C_VEL
LIN {X 0,Y 439.57,Z 447.362,A -85,B 0,C 180,E1 -9101.061,E2 -9101.061} C_VEL
LIN {X 0,Y 440.06,Z 440.436,A -85,B 0,C 180,E1 -9101.983,E2 -9101.983} C_VEL
LIN {X 0,Y 440.562,Z 432.254,A -85,B 0,C 180,E1 -9102.905,E2 -9102.905} C_VEL
LIN {X 0,Y 441.016,Z 424.259,A -85,B 0,C 180,E1 -9103.667,E2 -9103.667} C_VEL
LIN {X 0,Y 441.545,Z 415.022,A -85,B 0,C 180,E1 -9104.401,E2 -9104.401} C_VEL
LIN {X 0,Y 442.051,Z 405.262,A -85,B 0,C 180,E1 -9105.031,E2 -9105.031} C_VEL
LIN {X 0,Y 442.528,Z 395.179,A -85,B 0,C 180,E1 -9105.545,E2 -9105.545} C_VEL
LIN {X 0,Y 442.968,Z 385.665,A -85,B 0,C 180,E1 -9105.913,E2 -9105.913} C_VEL
LIN {X 0,Y 443.247,Z 376.683,A -85,B 0,C 180,E1 -9106.169,E2 -9106.169} C_VEL
LIN {X 0,Y 443.495,Z 351.676,A -85,B 0,C 180,E1 -9106.609,E2 -9106.609} C_VEL
LIN {X 0,Y 443.901,Z 291.65,A -85,B 0,C 180,E1 -9107.588,E2 -9107.588} C_VEL
LIN {X 0,Y 439.989,Z 269.475,A -85,B 0,C 180,E1 -9108.141,E2 -9108.141} C_VEL
LIN {X 0,Y 439.978,Z 268.722,A -85,B 0,C 180,E1 -9108.233,E2 -9108.233} C_VEL
LIN {X 0,Y 440.752,Z 255.193,A -85,B 0,C 180,E1 -9111.515,E2 -9111.515} C_VEL
LIN {X 0,Y 441.629,Z 240.918,A -85,B 0,C 180,E1 -9114.893,E2 -9114.893} C_VEL
LIN {X 0,Y 440.835,Z 234.488,A -85,B 0,C 180,E1 -9116.512,E2 -9116.512} C_VEL
LIN {X 0,Y 439.44,Z 227.272,A -85,B 0,C 180,E1 -9118.493,E2 -9118.493} C_VEL
LIN {X 0,Y 439.372,Z 227.251,A -85,B 0,C 180,E1 -9122.03,E2 -9122.03} C_VEL
LIN {X 0,Y 439.396,Z 227.245,A -85,B 0,C 180,E1 -9125.34,E2 -9125.34} C_VEL
LIN {X 0,Y 439.385,Z 227.249,A -85,B 0,C 180,E1 -9128.595,E2 -9128.595} C_VEL
LIN {X 0,Y 439.39,Z 227.238,A -85,B 0,C 180,E1 -9131.256,E2 -9131.256} C_VEL
LIN {X 0,Y 439.401,Z 227.246,A -85,B 0,C 180,E1 -9134.729,E2 -9134.729} C_VEL
LIN {X 0,Y 439.397,Z 227.253,A -85,B 0,C 180,E1 -9137.795,E2 -9137.795} C_VEL
LIN {X 0,Y 439.396,Z 227.244,A -85,B 0,C 180,E1 -9140.223,E2 -9140.223} C_VEL
LIN {X 0,Y 439.374,Z 227.253,A -85,B 0,C 180,E1 -9143.712,E2 -9143.712} C_VEL
LIN {X 0,Y 439.37,Z 227.245,A -85,B 0,C 180,E1 -9147.053,E2 -9147.053} C_VEL
LIN {X 0,Y 439.382,Z 227.249,A -85,B 0,C 180,E1 -9150.274,E2 -9150.274} C_VEL
LIN {X 0,Y 439.429,Z 227.235,A -85,B 0,C 180,E1 -9153.396,E2 -9153.396} C_VEL
LIN {X 0,Y 439.386,Z 227.248,A -85,B 0,C 180,E1 -9156.429,E2 -9156.429} C_VEL
LIN {X 0,Y 439.388,Z 227.243,A -85,B 0,C 180,E1 -9159.397,E2 -9159.397} C_VEL
LIN {X 0,Y 439.405,Z 227.233,A -85,B 0,C 180,E1 -9162.308,E2 -9162.308} C_VEL
LIN {X 0,Y 439.448,Z 227.247,A -85,B 0,C 180,E1 -9165.173,E2 -9165.173} C_VEL
LIN {X 0,Y 439.483,Z 227.231,A -85,B 0,C 180,E1 -9168.001,E2 -9168.001} C_VEL
LIN {X 0,Y 439.503,Z 227.225,A -85,B 0,C 180,E1 -9171.725,E2 -9171.725} C_VEL
LIN {X 0,Y 439.611,Z 227.223,A -85,B 0,C 180,E1 -9174.495,E2 -9174.495} C_VEL
LIN {X 0,Y 439.634,Z 227.214,A -85,B 0,C 180,E1 -9178.167,E2 -9178.167} C_VEL
LIN {X 0,Y 439.762,Z 227.184,A -85,B 0,C 180,E1 -9179.999,E2 -9179.999} C_VEL
LIN {X 0,Y 439.654,Z 227.214,A -85,B 0,C 180,E1 -9182.748,E2 -9182.748} C_VEL
LIN {X 0,Y 439.61,Z 227.226,A -85,B 0,C 180,E1 -9186.425,E2 -9186.425} C_VEL
LIN {X 0,Y 439.499,Z 227.218,A -85,B 0,C 180,E1 -9189.201,E2 -9189.201} C_VEL
LIN {X 0,Y 439.464,Z 227.242,A -85,B 0,C 180,E1 -9192.937,E2 -9192.937} C_VEL
LIN {X 0,Y 439.446,Z 227.245,A -85,B 0,C 180,E1 -9196.348,E2 -9196.348} C_VEL
LIN {X 0,Y 439.4,Z 227.232,A -85,B 0,C 180,E1 -9199.626,E2 -9199.626} C_VEL
LIN {X 0,Y 439.361,Z 227.258,A -85,B 0,C 180,E1 -9202.575,E2 -9202.575} C_VEL
LIN {X 0,Y 439.395,Z 227.246,A -85,B 0,C 180,E1 -9205.585,E2 -9205.585} C_VEL
LIN {X 0,Y 439.414,Z 227.245,A -85,B 0,C 180,E1 -9208.673,E2 -9208.673} C_VEL
LIN {X 0,Y 439.368,Z 227.258,A -85,B 0,C 180,E1 -9212.03,E2 -9212.03} C_VEL
LIN {X 0,Y 439.392,Z 227.241,A -85,B 0,C 180,E1 -9215.34,E2 -9215.34} C_VEL
LIN {X 0,Y 439.387,Z 227.25,A -85,B 0,C 180,E1 -9218.594,E2 -9218.594} C_VEL
LIN {X 0,Y 439.387,Z 227.243,A -85,B 0,C 180,E1 -9221.257,E2 -9221.257} C_VEL
LIN {X 0,Y 439.405,Z 227.245,A -85,B 0,C 180,E1 -9224.728,E2 -9224.728} C_VEL
LIN {X 0,Y 439.393,Z 227.225,A -85,B 0,C 180,E1 -9227.796,E2 -9227.796} C_VEL
LIN {X 0,Y 439.445,Z 227.241,A -85,B 0,C 180,E1 -9230.23,E2 -9230.23} C_VEL
LIN {X 0,Y 439.373,Z 227.248,A -85,B 0,C 180,E1 -9233.713,E2 -9233.713} C_VEL
LIN {X 0,Y 439.368,Z 227.249,A -85,B 0,C 180,E1 -9237.054,E2 -9237.054} C_VEL
LIN {X 0,Y 439.378,Z 227.24,A -85,B 0,C 180,E1 -9240.274,E2 -9240.274} C_VEL
LIN {X 0,Y 439.426,Z 227.251,A -85,B 0,C 180,E1 -9243.396,E2 -9243.396} C_VEL
LIN {X 0,Y 439.382,Z 227.253,A -85,B 0,C 180,E1 -9246.429,E2 -9246.429} C_VEL
LIN {X 0,Y 439.385,Z 227.257,A -85,B 0,C 180,E1 -9249.397,E2 -9249.397} C_VEL
LIN {X 0,Y 439.428,Z 227.248,A -85,B 0,C 180,E1 -9252.309,E2 -9252.309} C_VEL
LIN {X 0,Y 439.446,Z 227.249,A -85,B 0,C 180,E1 -9255.174,E2 -9255.174} C_VEL
LIN {X 0,Y 439.48,Z 227.243,A -85,B 0,C 180,E1 -9258.001,E2 -9258.001} C_VEL
LIN {X 0,Y 439.544,Z 227.235,A -85,B 0,C 180,E1 -9261.726,E2 -9261.726} C_VEL
LIN {X 0,Y 439.619,Z 227.226,A -85,B 0,C 180,E1 -9264.496,E2 -9264.496} C_VEL
LIN {X 0,Y 439.633,Z 227.223,A -85,B 0,C 180,E1 -9268.168,E2 -9268.168} C_VEL
LIN {X 0,Y 439.761,Z 227.208,A -85,B 0,C 180,E1 -9270,E2 -9270} C_VEL
LIN {X 0,Y 439.619,Z 227.226,A -85,B 0,C 180,E1 -9270.989,E2 -9270.989} C_VEL
LIN {X 0,Y 438.902,Z 227.314,A -85,B 0,C 180,E1 -9271.753,E2 -9271.753} C_VEL
LIN {X 0,Y 435.924,Z 227.687,A -85,B 0,C 180,E1 -9272.992,E2 -9272.992} C_VEL
LIN {X 0,Y 433.472,Z 227.993,A -85,B 0,C 180,E1 -9273.992,E2 -9273.992} C_VEL
LIN {X 0,Y 432.499,Z 228.114,A -85,B 0,C 180,E1 -9274.767,E2 -9274.767} C_VEL
LIN {X 0,Y 432.462,Z 228.116,A -85,B 0,C 180,E1 -9275.029,E2 -9275.029} C_VEL
LIN {X 0,Y 432.582,Z 228.102,A -85,B 0,C 180,E1 -9277.679,E2 -9277.679} C_VEL
LIN {X 0,Y 432.39,Z 228.126,A -85,B 0,C 180,E1 -9281.247,E2 -9281.247} C_VEL
LIN {X 0,Y 432.371,Z 228.129,A -85,B 0,C 180,E1 -9284.112,E2 -9284.112} C_VEL
LIN {X 0,Y 432.394,Z 228.126,A -85,B 0,C 180,E1 -9287.012,E2 -9287.012} C_VEL
LIN {X 0,Y 432.335,Z 228.132,A -85,B 0,C 180,E1 -9289.96,E2 -9289.96} C_VEL
LIN {X 0,Y 432.315,Z 228.136,A -85,B 0,C 180,E1 -9292.964,E2 -9292.964} C_VEL
LIN {X 0,Y 432.36,Z 228.13,A -85,B 0,C 180,E1 -9296.033,E2 -9296.033} C_VEL
LIN {X 0,Y 432.339,Z 228.114,A -85,B 0,C 180,E1 -9299.188,E2 -9299.188} C_VEL
LIN {X 0,Y 432.319,Z 228.132,A -85,B 0,C 180,E1 -9302.443,E2 -9302.443} C_VEL
LIN {X 0,Y 432.341,Z 228.116,A -85,B 0,C 180,E1 -9305.632,E2 -9305.632} C_VEL
LIN {X 0,Y 432.354,Z 228.126,A -85,B 0,C 180,E1 -9308.718,E2 -9308.718} C_VEL
LIN {X 0,Y 432.362,Z 228.1,A -85,B 0,C 180,E1 -9311.794,E2 -9311.794} C_VEL
LIN {X 0,Y 432.375,Z 228.123,A -85,B 0,C 180,E1 -9315.659,E2 -9315.659} C_VEL
LIN {X 0,Y 432.368,Z 228.119,A -85,B 0,C 180,E1 -9318.393,E2 -9318.393} C_VEL
LIN {X 0,Y 432.347,Z 228.132,A -85,B 0,C 180,E1 -9321.852,E2 -9321.852} C_VEL
LIN {X 0,Y 432.337,Z 228.121,A -85,B 0,C 180,E1 -9325.323,E2 -9325.323} C_VEL
LIN {X 0,Y 432.318,Z 228.131,A -85,B 0,C 180,E1 -9328.654,E2 -9328.654} C_VEL
LIN {X 0,Y 432.378,Z 228.112,A -85,B 0,C 180,E1 -9331.877,E2 -9331.877} C_VEL
LIN {X 0,Y 432.343,Z 228.124,A -85,B 0,C 180,E1 -9334.999,E2 -9334.999} C_VEL
LIN {X 0,Y 432.355,Z 228.124,A -85,B 0,C 180,E1 -9338.046,E2 -9338.046} C_VEL
LIN {X 0,Y 432.384,Z 228.106,A -85,B 0,C 180,E1 -9341.03,E2 -9341.03} C_VEL
LIN {X 0,Y 432.429,Z 228.118,A -85,B 0,C 180,E1 -9343.962,E2 -9343.962} C_VEL
LIN {X 0,Y 432.458,Z 228.106,A -85,B 0,C 180,E1 -9347.804,E2 -9347.804} C_VEL
LIN {X 0,Y 432.491,Z 228.101,A -85,B 0,C 180,E1 -9351.591,E2 -9351.591} C_VEL
LIN {X 0,Y 432.593,Z 228.096,A -85,B 0,C 180,E1 -9354.407,E2 -9354.407} C_VEL
LIN {X 0,Y 432.604,Z 228.084,A -85,B 0,C 180,E1 -9358.139,E2 -9358.139} C_VEL
LIN {X 0,Y 432.731,Z 228.06,A -85,B 0,C 180,E1 -9360.001,E2 -9360.001} C_VEL
LIN {X 0,Y 432.592,Z 228.093,A -85,B 0,C 180,E1 -9362.794,E2 -9362.794} C_VEL
LIN {X 0,Y 432.586,Z 228.097,A -85,B 0,C 180,E1 -9365.595,E2 -9365.595} C_VEL
LIN {X 0,Y 432.463,Z 228.102,A -85,B 0,C 180,E1 -9368.411,E2 -9368.411} C_VEL
LIN {X 0,Y 432.459,Z 228.106,A -85,B 0,C 180,E1 -9372.197,E2 -9372.197} C_VEL
LIN {X 0,Y 432.43,Z 228.112,A -85,B 0,C 180,E1 -9376.039,E2 -9376.039} C_VEL
LIN {X 0,Y 432.386,Z 228.111,A -85,B 0,C 180,E1 -9379.485,E2 -9379.485} C_VEL
LIN {X 0,Y 432.319,Z 228.133,A -85,B 0,C 180,E1 -9382.965,E2 -9382.965} C_VEL
LIN {X 0,Y 432.363,Z 228.117,A -85,B 0,C 180,E1 -9386.033,E2 -9386.033} C_VEL
LIN {X 0,Y 432.343,Z 228.127,A -85,B 0,C 180,E1 -9389.188,E2 -9389.188} C_VEL
LIN {X 0,Y 432.321,Z 228.13,A -85,B 0,C 180,E1 -9392.444,E2 -9392.444} C_VEL
LIN {X 0,Y 432.338,Z 228.125,A -85,B 0,C 180,E1 -9395.818,E2 -9395.818} C_VEL
LIN {X 0,Y 432.328,Z 228.124,A -85,B 0,C 180,E1 -9399.346,E2 -9399.346} C_VEL
LIN {X 0,Y 432.334,Z 228.128,A -85,B 0,C 180,E1 -9401.798,E2 -9401.798} C_VEL
LIN {X 0,Y 432.335,Z 228.128,A -85,B 0,C 180,E1 -9404.348,E2 -9404.348} C_VEL
LIN {X 0,Y 432.322,Z 228.131,A -85,B 0,C 180,E1 -9407.016,E2 -9407.016} C_VEL
LIN {X 0,Y 432.338,Z 228.115,A -85,B 0,C 180,E1 -9409.821,E2 -9409.821} C_VEL
LIN {X 0,Y 432.309,Z 228.131,A -85,B 0,C 180,E1 -9413.022,E2 -9413.022} C_VEL
LIN {X 0,Y 432.361,Z 228.13,A -85,B 0,C 180,E1 -9415.997,E2 -9415.997} C_VEL
LIN {X 0,Y 432.349,Z 228.131,A -85,B 0,C 180,E1 -9419.49,E2 -9419.49} C_VEL
LIN {X 0,Y 432.447,Z 228.309,A -85,B 0,C 180,E1 -9421.354,E2 -9421.354} C_VEL
LIN {X 0,Y 434.265,Z 238.321,A -85,B 0,C 180,E1 -9424.09,E2 -9424.09} C_VEL
LIN {X 0,Y 434.559,Z 242.378,A -85,B 0,C 180,E1 -9425.135,E2 -9425.135} C_VEL
LIN {X 0,Y 433.7,Z 256.876,A -85,B 0,C 180,E1 -9428.617,E2 -9428.617} C_VEL
LIN {X 0,Y 433.03,Z 267.872,A -85,B 0,C 180,E1 -9431.305,E2 -9431.305} C_VEL
LIN {X 0,Y 433.004,Z 269.188,A -85,B 0,C 180,E1 -9431.549,E2 -9431.549} C_VEL
LIN {X 0,Y 437.155,Z 292.809,A -85,B 0,C 180,E1 -9432.154,E2 -9432.154} C_VEL
LIN {X 0,Y 436.45,Z 373.826,A -85,B 0,C 180,E1 -9433.512,E2 -9433.512} C_VEL
LIN {X 0,Y 436.19,Z 383.723,A -85,B 0,C 180,E1 -9433.773,E2 -9433.773} C_VEL
LIN {X 0,Y 435.791,Z 393.699,A -85,B 0,C 180,E1 -9434.148,E2 -9434.148} C_VEL
LIN {X 0,Y 435.321,Z 403.055,A -85,B 0,C 180,E1 -9434.611,E2 -9434.611} C_VEL
LIN {X 0,Y 434.769,Z 413.198,A -85,B 0,C 180,E1 -9435.25,E2 -9435.25} C_VEL
LIN {X 0,Y 434.196,Z 422.195,A -85,B 0,C 180,E1 -9435.949,E2 -9435.949} C_VEL
LIN {X 0,Y 433.688,Z 430.747,A -85,B 0,C 180,E1 -9436.749,E2 -9436.749} C_VEL
LIN {X 0,Y 433.241,Z 438.323,A -85,B 0,C 180,E1 -9437.588,E2 -9437.588} C_VEL
LIN {X 0,Y 432.726,Z 445.543,A -85,B 0,C 180,E1 -9438.524,E2 -9438.524} C_VEL
LIN {X 0,Y 432.321,Z 451.745,A -85,B 0,C 180,E1 -9439.462,E2 -9439.462} C_VEL
LIN {X 0,Y 431.938,Z 458.283,A -85,B 0,C 180,E1 -9440.636,E2 -9440.636} C_VEL
LIN {X 0,Y 431.683,Z 462.785,A -85,B 0,C 180,E1 -9441.574,E2 -9441.574} C_VEL
LIN {X 0,Y 431.417,Z 468.275,A -85,B 0,C 180,E1 -9442.982,E2 -9442.982} C_VEL
LIN {X 0,Y 431.277,Z 472.598,A -85,B 0,C 180,E1 -9444.389,E2 -9444.389} C_VEL
LIN {X 0,Y 431.271,Z 474.965,A -85,B 0,C 180,E1 -9445.326,E2 -9445.326} C_VEL
LIN {X 0,Y 431.236,Z 478.147,A -85,B 0,C 180,E1 -9447.198,E2 -9447.198} C_VEL
LIN {X 0,Y 431.203,Z 479.203,A -85,B 0,C 180,E1 -9448.132,E2 -9448.132} C_VEL
LIN {X 0,Y 431.169,Z 479.79,A -85,B 0,C 180,E1 -9449.066,E2 -9449.066} C_VEL
LIN {X 0,Y 431.169,Z 479.79,A -85,B 0,C 180,E1 -9450.934,E2 -9450.934} C_VEL
LIN {X 0,Y 431.203,Z 479.203,A -85,B 0,C 180,E1 -9451.868,E2 -9451.868} C_VEL
LIN {X 0,Y 431.188,Z 476.76,A -85,B 0,C 180,E1 -9453.738,E2 -9453.738} C_VEL
LIN {X 0,Y 431.293,Z 473.815,A -85,B 0,C 180,E1 -9455.142,E2 -9455.142} C_VEL
LIN {X 0,Y 431.377,Z 469.829,A -85,B 0,C 180,E1 -9456.548,E2 -9456.548} C_VEL
LIN {X 0,Y 431.566,Z 464.7,A -85,B 0,C 180,E1 -9457.956,E2 -9457.956} C_VEL
LIN {X 0,Y 431.844,Z 459.438,A -85,B 0,C 180,E1 -9459.13,E2 -9459.13} C_VEL
LIN {X 0,Y 432.225,Z 453.121,A -85,B 0,C 180,E1 -9460.303,E2 -9460.303} C_VEL
LIN {X 0,Y 432.585,Z 447.169,A -85,B 0,C 180,E1 -9461.242,E2 -9461.242} C_VEL
LIN {X 0,Y 433.088,Z 440.242,A -85,B 0,C 180,E1 -9462.179,E2 -9462.179} C_VEL
LIN {X 0,Y 433.623,Z 432.061,A -85,B 0,C 180,E1 -9463.115,E2 -9463.115} C_VEL
LIN {X 0,Y 434.119,Z 423.368,A -85,B 0,C 180,E1 -9463.95,E2 -9463.95} C_VEL
LIN {X 0,Y 434.656,Z 414.829,A -85,B 0,C 180,E1 -9464.634,E2 -9464.634} C_VEL
LIN {X 0,Y 435.214,Z 405.069,A -85,B 0,C 180,E1 -9465.273,E2 -9465.273} C_VEL
LIN {X 0,Y 435.642,Z 396.274,A -85,B 0,C 180,E1 -9465.737,E2 -9465.737} C_VEL
LIN {X 0,Y 436.111,Z 386.346,A -85,B 0,C 180,E1 -9466.14,E2 -9466.14} C_VEL
LIN {X 0,Y 436.436,Z 376.49,A -85,B 0,C 180,E1 -9466.428,E2 -9466.428} C_VEL
LIN {X 0,Y 436.7,Z 351.582,A -85,B 0,C 180,E1 -9466.874,E2 -9466.874} C_VEL
LIN {X 0,Y 437.198,Z 292.842,A -85,B 0,C 180,E1 -9467.844,E2 -9467.844} C_VEL
LIN {X 0,Y 433.03,Z 269.248,A -85,B 0,C 180,E1 -9468.445,E2 -9468.445} C_VEL
LIN {X 0,Y 433.022,Z 267.966,A -85,B 0,C 180,E1 -9468.671,E2 -9468.671} C_VEL
LIN {X 0,Y 433.826,Z 255.028,A -85,B 0,C 180,E1 -9471.876,E2 -9471.876} C_VEL
LIN {X 0,Y 434.694,Z 241.581,A -85,B 0,C 180,E1 -9475.123,E2 -9475.123} C_VEL
LIN {X 0,Y 433.428,Z 233.332,A -85,B 0,C 180,E1 -9477.263,E2 -9477.263} C_VEL
LIN {X 0,Y 432.404,Z 228.144,A -85,B 0,C 180,E1 -9478.744,E2 -9478.744} C_VEL
LIN {X 0,Y 432.327,Z 228.127,A -85,B 0,C 180,E1 -9482.293,E2 -9482.293} C_VEL
LIN {X 0,Y 432.342,Z 228.127,A -85,B 0,C 180,E1 -9484.677,E2 -9484.677} C_VEL
LIN {X 0,Y 432.341,Z 228.13,A -85,B 0,C 180,E1 -9488.149,E2 -9488.149} C_VEL
LIN {X 0,Y 432.334,Z 228.12,A -85,B 0,C 180,E1 -9491.602,E2 -9491.602} C_VEL
LIN {X 0,Y 432.335,Z 228.128,A -85,B 0,C 180,E1 -9494.347,E2 -9494.347} C_VEL
LIN {X 0,Y 432.321,Z 228.13,A -85,B 0,C 180,E1 -9497.015,E2 -9497.015} C_VEL
LIN {X 0,Y 432.334,Z 228.125,A -85,B 0,C 180,E1 -9499.82,E2 -9499.82} C_VEL
LIN {X 0,Y 432.307,Z 228.134,A -85,B 0,C 180,E1 -9503.022,E2 -9503.022} C_VEL
LIN {X 0,Y 432.333,Z 228.12,A -85,B 0,C 180,E1 -9506.001,E2 -9506.001} C_VEL
LIN {X 0,Y 432.348,Z 228.132,A -85,B 0,C 180,E1 -9509.489,E2 -9509.489} C_VEL
LIN {X 0,Y 432.391,Z 228.111,A -85,B 0,C 180,E1 -9512.928,E2 -9512.928} C_VEL
LIN {X 0,Y 432.37,Z 228.123,A -85,B 0,C 180,E1 -9516.023,E2 -9516.023} C_VEL
LIN {X 0,Y 432.35,Z 228.125,A -85,B 0,C 180,E1 -9519.046,E2 -9519.046} C_VEL
LIN {X 0,Y 432.361,Z 228.11,A -85,B 0,C 180,E1 -9522.01,E2 -9522.01} C_VEL
LIN {X 0,Y 432.395,Z 228.122,A -85,B 0,C 180,E1 -9524.926,E2 -9524.926} C_VEL
LIN {X 0,Y 432.459,Z 228.106,A -85,B 0,C 180,E1 -9527.803,E2 -9527.803} C_VEL
LIN {X 0,Y 432.463,Z 228.102,A -85,B 0,C 180,E1 -9531.589,E2 -9531.589} C_VEL
LIN {X 0,Y 432.586,Z 228.097,A -85,B 0,C 180,E1 -9534.405,E2 -9534.405} C_VEL
LIN {X 0,Y 432.604,Z 228.089,A -85,B 0,C 180,E1 -9538.138,E2 -9538.138} C_VEL
LIN {X 0,Y 432.731,Z 228.06,A -85,B 0,C 180,E1 -9539.999,E2 -9539.999} C_VEL
LIN {X 0,Y 432.603,Z 228.092,A -85,B 0,C 180,E1 -9542.793,E2 -9542.793} C_VEL
LIN {X 0,Y 432.564,Z 228.104,A -85,B 0,C 180,E1 -9546.53,E2 -9546.53} C_VEL
LIN {X 0,Y 432.441,Z 228.096,A -85,B 0,C 180,E1 -9549.353,E2 -9549.353} C_VEL
LIN {X 0,Y 432.429,Z 228.119,A -85,B 0,C 180,E1 -9552.803,E2 -9552.803} C_VEL
LIN {X 0,Y 432.411,Z 228.119,A -85,B 0,C 180,E1 -9556.478,E2 -9556.478} C_VEL
LIN {X 0,Y 432.336,Z 228.113,A -85,B 0,C 180,E1 -9559.96,E2 -9559.96} C_VEL
LIN {X 0,Y 432.315,Z 228.132,A -85,B 0,C 180,E1 -9562.964,E2 -9562.964} C_VEL
LIN {X 0,Y 432.358,Z 228.122,A -85,B 0,C 180,E1 -9566.032,E2 -9566.032} C_VEL
LIN {X 0,Y 432.34,Z 228.124,A -85,B 0,C 180,E1 -9569.187,E2 -9569.187} C_VEL
LIN {X 0,Y 432.32,Z 228.13,A -85,B 0,C 180,E1 -9572.443,E2 -9572.443} C_VEL
LIN {X 0,Y 432.342,Z 228.121,A -85,B 0,C 180,E1 -9575.632,E2 -9575.632} C_VEL
LIN {X 0,Y 432.349,Z 228.126,A -85,B 0,C 180,E1 -9578.716,E2 -9578.716} C_VEL
LIN {X 0,Y 432.363,Z 228.122,A -85,B 0,C 180,E1 -9581.793,E2 -9581.793} C_VEL
LIN {X 0,Y 432.375,Z 228.123,A -85,B 0,C 180,E1 -9584.341,E2 -9584.341} C_VEL
LIN {X 0,Y 432.363,Z 228.101,A -85,B 0,C 180,E1 -9588.393,E2 -9588.393} C_VEL
LIN {X 0,Y 432.347,Z 228.134,A -85,B 0,C 180,E1 -9591.851,E2 -9591.851} C_VEL
LIN {X 0,Y 432.337,Z 228.113,A -85,B 0,C 180,E1 -9595.323,E2 -9595.323} C_VEL
LIN {X 0,Y 432.318,Z 228.132,A -85,B 0,C 180,E1 -9598.654,E2 -9598.654} C_VEL
LIN {X 0,Y 432.379,Z 228.122,A -85,B 0,C 180,E1 -9601.877,E2 -9601.877} C_VEL
LIN {X 0,Y 432.348,Z 228.131,A -85,B 0,C 180,E1 -9604.999,E2 -9604.999} C_VEL
LIN {X 0,Y 432.354,Z 228.13,A -85,B 0,C 180,E1 -9608.046,E2 -9608.046} C_VEL
LIN {X 0,Y 432.383,Z 228.128,A -85,B 0,C 180,E1 -9611.03,E2 -9611.03} C_VEL
LIN {X 0,Y 432.427,Z 228.121,A -85,B 0,C 180,E1 -9613.961,E2 -9613.961} C_VEL
LIN {X 0,Y 432.456,Z 228.118,A -85,B 0,C 180,E1 -9617.803,E2 -9617.803} C_VEL
LIN {X 0,Y 432.488,Z 228.114,A -85,B 0,C 180,E1 -9621.59,E2 -9621.59} C_VEL
LIN {X 0,Y 432.596,Z 228.101,A -85,B 0,C 180,E1 -9624.406,E2 -9624.406} C_VEL
LIN {X 0,Y 432.603,Z 228.099,A -85,B 0,C 180,E1 -9628.138,E2 -9628.138} C_VEL
LIN {X 0,Y 432.73,Z 228.084,A -85,B 0,C 180,E1 -9630,E2 -9630} C_VEL
LIN {X 0,Y 432.602,Z 228.1,A -85,B 0,C 180,E1 -9632.794,E2 -9632.794} C_VEL
LIN {X 0,Y 432.462,Z 228.116,A -85,B 0,C 180,E1 -9635.029,E2 -9635.029} C_VEL
LIN {X 0,Y 431.903,Z 228.187,A -85,B 0,C 180,E1 -9635.807,E2 -9635.807} C_VEL
LIN {X 0,Y 429.056,Z 228.543,A -85,B 0,C 180,E1 -9637.072,E2 -9637.072} C_VEL
LIN {X 0,Y 426.572,Z 228.852,A -85,B 0,C 180,E1 -9638.093,E2 -9638.093} C_VEL
LIN {X 0,Y 425.49,Z 228.987,A -85,B 0,C 180,E1 -9638.883,E2 -9638.883} C_VEL
LIN {X 0,Y 425.399,Z 228.996,A -85,B 0,C 180,E1 -9639.151,E2 -9639.151} C_VEL
LIN {X 0,Y 425.39,Z 228.999,A -85,B 0,C 180,E1 -9642.904,E2 -9642.904} C_VEL
LIN {X 0,Y 425.358,Z 229.003,A -85,B 0,C 180,E1 -9646.605,E2 -9646.605} C_VEL
LIN {X 0,Y 425.325,Z 229.005,A -85,B 0,C 180,E1 -9649.636,E2 -9649.636} C_VEL
LIN {X 0,Y 425.303,Z 229.007,A -85,B 0,C 180,E1 -9653.365,E2 -9653.365} C_VEL
LIN {X 0,Y 425.344,Z 229.004,A -85,B 0,C 180,E1 -9656.845,E2 -9656.845} C_VEL
LIN {X 0,Y 425.287,Z 228.993,A -85,B 0,C 180,E1 -9659.72,E2 -9659.72} C_VEL
LIN {X 0,Y 425.278,Z 229.003,A -85,B 0,C 180,E1 -9663.048,E2 -9663.048} C_VEL
LIN {X 0,Y 425.281,Z 228.997,A -85,B 0,C 180,E1 -9665.929,E2 -9665.929} C_VEL
LIN {X 0,Y 425.307,Z 229.002,A -85,B 0,C 180,E1 -9669.046,E2 -9669.046} C_VEL
LIN {X 0,Y 425.311,Z 228.977,A -85,B 0,C 180,E1 -9671.962,E2 -9671.962} C_VEL
LIN {X 0,Y 425.309,Z 229,A -85,B 0,C 180,E1 -9675.279,E2 -9675.279} C_VEL
LIN {X 0,Y 425.304,Z 228.997,A -85,B 0,C 180,E1 -9678.626,E2 -9678.626} C_VEL
LIN {X 0,Y 425.318,Z 229.001,A -85,B 0,C 180,E1 -9681.104,E2 -9681.104} C_VEL
LIN {X 0,Y 425.297,Z 228.997,A -85,B 0,C 180,E1 -9684.665,E2 -9684.665} C_VEL
LIN {X 0,Y 425.263,Z 229.014,A -85,B 0,C 180,E1 -9688.074,E2 -9688.074} C_VEL
LIN {X 0,Y 425.328,Z 228.999,A -85,B 0,C 180,E1 -9691.368,E2 -9691.368} C_VEL
LIN {X 0,Y 425.351,Z 228.986,A -85,B 0,C 180,E1 -9693.506,E2 -9693.506} C_VEL
LIN {X 0,Y 425.282,Z 229.007,A -85,B 0,C 180,E1 -9696.634,E2 -9696.634} C_VEL
LIN {X 0,Y 425.293,Z 228.994,A -85,B 0,C 180,E1 -9699.695,E2 -9699.695} C_VEL
LIN {X 0,Y 425.34,Z 228.992,A -85,B 0,C 180,E1 -9702.698,E2 -9702.698} C_VEL
LIN {X 0,Y 425.348,Z 229.003,A -85,B 0,C 180,E1 -9705.651,E2 -9705.651} C_VEL
LIN {X 0,Y 425.35,Z 228.988,A -85,B 0,C 180,E1 -9708.565,E2 -9708.565} C_VEL
LIN {X 0,Y 425.537,Z 228.969,A -85,B 0,C 180,E1 -9712.408,E2 -9712.408} C_VEL
LIN {X 0,Y 425.549,Z 228.973,A -85,B 0,C 180,E1 -9714.314,E2 -9714.314} C_VEL
LIN {X 0,Y 425.574,Z 228.959,A -85,B 0,C 180,E1 -9718.108,E2 -9718.108} C_VEL
LIN {X 0,Y 425.701,Z 228.935,A -85,B 0,C 180,E1 -9720.001,E2 -9720.001} C_VEL
LIN {X 0,Y 425.546,Z 228.971,A -85,B 0,C 180,E1 -9722.84,E2 -9722.84} C_VEL
LIN {X 0,Y 425.541,Z 228.974,A -85,B 0,C 180,E1 -9725.687,E2 -9725.687} C_VEL
LIN {X 0,Y 425.407,Z 228.98,A -85,B 0,C 180,E1 -9728.551,E2 -9728.551} C_VEL
LIN {X 0,Y 425.412,Z 228.985,A -85,B 0,C 180,E1 -9732.402,E2 -9732.402} C_VEL
LIN {X 0,Y 425.388,Z 228.991,A -85,B 0,C 180,E1 -9736.312,E2 -9736.312} C_VEL
LIN {X 0,Y 425.328,Z 228.989,A -85,B 0,C 180,E1 -9739.636,E2 -9739.636} C_VEL
LIN {X 0,Y 425.288,Z 229.006,A -85,B 0,C 180,E1 -9742.339,E2 -9742.339} C_VEL
LIN {X 0,Y 425.293,Z 228.996,A -85,B 0,C 180,E1 -9745.446,E2 -9745.446} C_VEL
LIN {X 0,Y 425.332,Z 228.997,A -85,B 0,C 180,E1 -9748.633,E2 -9748.633} C_VEL
LIN {X 0,Y 425.263,Z 229.009,A -85,B 0,C 180,E1 -9751.928,E2 -9751.928} C_VEL
LIN {X 0,Y 425.296,Z 229.001,A -85,B 0,C 180,E1 -9755.337,E2 -9755.337} C_VEL
LIN {X 0,Y 425.298,Z 229.001,A -85,B 0,C 180,E1 -9758.899,E2 -9758.899} C_VEL
LIN {X 0,Y 425.291,Z 229.007,A -85,B 0,C 180,E1 -9761.959,E2 -9761.959} C_VEL
LIN {X 0,Y 425.286,Z 229.005,A -85,B 0,C 180,E1 -9765.284,E2 -9765.284} C_VEL
LIN {X 0,Y 425.276,Z 228.997,A -85,B 0,C 180,E1 -9768.622,E2 -9768.622} C_VEL
LIN {X 0,Y 425.312,Z 229.002,A -85,B 0,C 180,E1 -9771.103,E2 -9771.103} C_VEL
LIN {X 0,Y 425.301,Z 228.999,A -85,B 0,C 180,E1 -9774.664,E2 -9774.664} C_VEL
LIN {X 0,Y 425.267,Z 229.008,A -85,B 0,C 180,E1 -9778.073,E2 -9778.073} C_VEL
LIN {X 0,Y 425.374,Z 229.155,A -85,B 0,C 180,E1 -9781.09,E2 -9781.09} C_VEL
LIN {X 0,Y 427.058,Z 238.18,A -85,B 0,C 180,E1 -9783.619,E2 -9783.619} C_VEL
LIN {X 0,Y 427.629,Z 243.244,A -85,B 0,C 180,E1 -9784.964,E2 -9784.964} C_VEL
LIN {X 0,Y 426.725,Z 257.744,A -85,B 0,C 180,E1 -9788.503,E2 -9788.503} C_VEL
LIN {X 0,Y 426.047,Z 268.716,A -85,B 0,C 180,E1 -9791.206,E2 -9791.206} C_VEL
LIN {X 0,Y 426.618,Z 272.102,A -85,B 0,C 180,E1 -9791.344,E2 -9791.344} C_VEL
LIN {X 0,Y 430.447,Z 294.224,A -85,B 0,C 180,E1 -9791.894,E2 -9791.894} C_VEL
LIN {X 0,Y 429.645,Z 373.633,A -85,B 0,C 180,E1 -9793.244,E2 -9793.244} C_VEL
LIN {X 0,Y 429.376,Z 383.53,A -85,B 0,C 180,E1 -9793.508,E2 -9793.508} C_VEL
LIN {X 0,Y 428.969,Z 393.507,A -85,B 0,C 180,E1 -9793.889,E2 -9793.889} C_VEL
LIN {X 0,Y 428.458,Z 402.862,A -85,B 0,C 180,E1 -9794.358,E2 -9794.358} C_VEL
LIN {X 0,Y 427.892,Z 413.004,A -85,B 0,C 180,E1 -9795.008,E2 -9795.008} C_VEL
LIN {X 0,Y 427.281,Z 422.001,A -85,B 0,C 180,E1 -9795.716,E2 -9795.716} C_VEL
LIN {X 0,Y 426.782,Z 429.996,A -85,B 0,C 180,E1 -9796.471,E2 -9796.471} C_VEL
LIN {X 0,Y 426.27,Z 438.129,A -85,B 0,C 180,E1 -9797.382,E2 -9797.382} C_VEL
LIN {X 0,Y 425.744,Z 445.349,A -85,B 0,C 180,E1 -9798.333,E2 -9798.333} C_VEL
LIN {X 0,Y 425.29,Z 451.551,A -85,B 0,C 180,E1 -9799.286,E2 -9799.286} C_VEL
LIN {X 0,Y 424.881,Z 458.089,A -85,B 0,C 180,E1 -9800.479,E2 -9800.479} C_VEL
LIN {X 0,Y 424.637,Z 462.591,A -85,B 0,C 180,E1 -9801.434,E2 -9801.434} C_VEL
LIN {X 0,Y 424.341,Z 468.081,A -85,B 0,C 180,E1 -9802.865,E2 -9802.865} C_VEL
LIN {X 0,Y 424.189,Z 472.405,A -85,B 0,C 180,E1 -9804.295,E2 -9804.295} C_VEL
LIN {X 0,Y 424.2,Z 474.772,A -85,B 0,C 180,E1 -9805.248,E2 -9805.248} C_VEL
LIN {X 0,Y 424.132,Z 477.954,A -85,B 0,C 180,E1 -9807.151,E2 -9807.151} C_VEL
LIN {X 0,Y 424.129,Z 479.011,A -85,B 0,C 180,E1 -9808.101,E2 -9808.101} C_VEL
LIN {X 0,Y 424.089,Z 479.598,A -85,B 0,C 180,E1 -9809.05,E2 -9809.05} C_VEL
LIN {X 0,Y 424.089,Z 479.598,A -85,B 0,C 180,E1 -9810.95,E2 -9810.95} C_VEL
LIN {X 0,Y 424.129,Z 479.011,A -85,B 0,C 180,E1 -9811.899,E2 -9811.899} C_VEL
LIN {X 0,Y 424.099,Z 476.567,A -85,B 0,C 180,E1 -9813.801,E2 -9813.801} C_VEL
LIN {X 0,Y 424.205,Z 473.622,A -85,B 0,C 180,E1 -9815.228,E2 -9815.228} C_VEL
LIN {X 0,Y 424.3,Z 469.635,A -85,B 0,C 180,E1 -9816.658,E2 -9816.658} C_VEL
LIN {X 0,Y 424.517,Z 464.506,A -85,B 0,C 180,E1 -9818.089,E2 -9818.089} C_VEL
LIN {X 0,Y 424.81,Z 459.245,A -85,B 0,C 180,E1 -9819.282,E2 -9819.282} C_VEL
LIN {X 0,Y 425.197,Z 452.927,A -85,B 0,C 180,E1 -9820.476,E2 -9820.476} C_VEL
LIN {X 0,Y 425.613,Z 446.976,A -85,B 0,C 180,E1 -9821.429,E2 -9821.429} C_VEL
LIN {X 0,Y 426.124,Z 440.048,A -85,B 0,C 180,E1 -9822.381,E2 -9822.381} C_VEL
LIN {X 0,Y 426.679,Z 431.868,A -85,B 0,C 180,E1 -9823.332,E2 -9823.332} C_VEL
LIN {X 0,Y 427.214,Z 423.092,A -85,B 0,C 180,E1 -9824.188,E2 -9824.188} C_VEL
LIN {X 0,Y 427.778,Z 414.636,A -85,B 0,C 180,E1 -9824.875,E2 -9824.875} C_VEL
LIN {X 0,Y 428.363,Z 404.877,A -85,B 0,C 180,E1 -9825.523,E2 -9825.523} C_VEL
LIN {X 0,Y 428.883,Z 394.794,A -85,B 0,C 180,E1 -9826.053,E2 -9826.053} C_VEL
LIN {X 0,Y 429.347,Z 385.28,A -85,B 0,C 180,E1 -9826.432,E2 -9826.432} C_VEL
LIN {X 0,Y 429.646,Z 376.298,A -85,B 0,C 180,E1 -9826.695,E2 -9826.695} C_VEL
LIN {X 0,Y 429.903,Z 351.493,A -85,B 0,C 180,E1 -9827.147,E2 -9827.147} C_VEL
LIN {X 0,Y 430.378,Z 293.361,A -85,B 0,C 180,E1 -9828.124,E2 -9828.124} C_VEL
LIN {X 0,Y 426.052,Z 268.985,A -85,B 0,C 180,E1 -9828.763,E2 -9828.763} C_VEL
LIN {X 0,Y 426.077,Z 267.682,A -85,B 0,C 180,E1 -9829.012,E2 -9829.012} C_VEL
LIN {X 0,Y 426.907,Z 254.862,A -85,B 0,C 180,E1 -9832.249,E2 -9832.249} C_VEL
LIN {X 0,Y 427.704,Z 242.328,A -85,B 0,C 180,E1 -9835.343,E2 -9835.343} C_VEL
LIN {X 0,Y 426.158,Z 233.187,A -85,B 0,C 180,E1 -9837.767,E2 -9837.767} C_VEL
LIN {X 0,Y 425.327,Z 229.027,A -85,B 0,C 180,E1 -9838.981,E2 -9838.981} C_VEL
LIN {X 0,Y 425.284,Z 229.005,A -85,B 0,C 180,E1 -9842.563,E2 -9842.563} C_VEL
LIN {X 0,Y 425.301,Z 229,A -85,B 0,C 180,E1 -9845.336,E2 -9845.336} C_VEL
LIN {X 0,Y 425.3,Z 229.004,A -85,B 0,C 180,E1 -9849.043,E2 -9849.043} C_VEL
LIN {X 0,Y 425.276,Z 229.007,A -85,B 0,C 180,E1 -9852.653,E2 -9852.653} C_VEL
LIN {X 0,Y 425.263,Z 229.011,A -85,B 0,C 180,E1 -9856.044,E2 -9856.044} C_VEL
LIN {X 0,Y 425.275,Z 229.006,A -85,B 0,C 180,E1 -9858.621,E2 -9858.621} C_VEL
LIN {X 0,Y 425.298,Z 229.001,A -85,B 0,C 180,E1 -9861.101,E2 -9861.101} C_VEL
LIN {X 0,Y 425.296,Z 229.001,A -85,B 0,C 180,E1 -9864.663,E2 -9864.663} C_VEL
LIN {X 0,Y 425.263,Z 229.009,A -85,B 0,C 180,E1 -9868.072,E2 -9868.072} C_VEL
LIN {X 0,Y 425.332,Z 228.997,A -85,B 0,C 180,E1 -9871.367,E2 -9871.367} C_VEL
LIN {X 0,Y 425.293,Z 228.996,A -85,B 0,C 180,E1 -9874.554,E2 -9874.554} C_VEL
LIN {X 0,Y 425.288,Z 229.006,A -85,B 0,C 180,E1 -9877.661,E2 -9877.661} C_VEL
LIN {X 0,Y 425.361,Z 228.985,A -85,B 0,C 180,E1 -9880.703,E2 -9880.703} C_VEL
LIN {X 0,Y 425.388,Z 228.991,A -85,B 0,C 180,E1 -9883.688,E2 -9883.688} C_VEL
LIN {X 0,Y 425.412,Z 228.985,A -85,B 0,C 180,E1 -9887.598,E2 -9887.598} C_VEL
LIN {X 0,Y 425.407,Z 228.98,A -85,B 0,C 180,E1 -9891.449,E2 -9891.449} C_VEL
LIN {X 0,Y 425.541,Z 228.974,A -85,B 0,C 180,E1 -9894.313,E2 -9894.313} C_VEL
LIN {X 0,Y 425.573,Z 228.965,A -85,B 0,C 180,E1 -9898.107,E2 -9898.107} C_VEL
LIN {X 0,Y 425.701,Z 228.935,A -85,B 0,C 180,E1 -9899.999,E2 -9899.999} C_VEL
LIN {X 0,Y 425.555,Z 228.97,A -85,B 0,C 180,E1 -9902.839,E2 -9902.839} C_VEL
LIN {X 0,Y 425.522,Z 228.979,A -85,B 0,C 180,E1 -9906.638,E2 -9906.638} C_VEL
LIN {X 0,Y 425.4,Z 228.972,A -85,B 0,C 180,E1 -9909.509,E2 -9909.509} C_VEL
LIN {X 0,Y 425.392,Z 228.995,A -85,B 0,C 180,E1 -9912.903,E2 -9912.903} C_VEL
LIN {X 0,Y 425.36,Z 228.995,A -85,B 0,C 180,E1 -9916.605,E2 -9916.605} C_VEL
LIN {X 0,Y 425.326,Z 228.984,A -85,B 0,C 180,E1 -9919.635,E2 -9919.635} C_VEL
LIN {X 0,Y 425.285,Z 229.009,A -85,B 0,C 180,E1 -9922.338,E2 -9922.338} C_VEL
LIN {X 0,Y 425.288,Z 229.002,A -85,B 0,C 180,E1 -9925.445,E2 -9925.445} C_VEL
LIN {X 0,Y 425.345,Z 228.983,A -85,B 0,C 180,E1 -9927.557,E2 -9927.557} C_VEL
LIN {X 0,Y 425.285,Z 229.008,A -85,B 0,C 180,E1 -9930.816,E2 -9930.816} C_VEL
LIN {X 0,Y 425.308,Z 228.996,A -85,B 0,C 180,E1 -9934.288,E2 -9934.288} C_VEL
LIN {X 0,Y 425.283,Z 229.01,A -85,B 0,C 180,E1 -9937.693,E2 -9937.693} C_VEL
LIN {X 0,Y 425.281,Z 229,A -85,B 0,C 180,E1 -9940.521,E2 -9940.521} C_VEL
LIN {X 0,Y 425.328,Z 229.003,A -85,B 0,C 180,E1 -9943.361,E2 -9943.361} C_VEL
LIN {X 0,Y 425.253,Z 228.992,A -85,B 0,C 180,E1 -9946.649,E2 -9946.649} C_VEL
LIN {X 0,Y 425.294,Z 228.989,A -85,B 0,C 180,E1 -9949.477,E2 -9949.477} C_VEL
LIN {X 0,Y 425.282,Z 229.008,A -85,B 0,C 180,E1 -9952.487,E2 -9952.487} C_VEL
LIN {X 0,Y 425.304,Z 228.99,A -85,B 0,C 180,E1 -9955.817,E2 -9955.817} C_VEL
LIN {X 0,Y 425.287,Z 229.008,A -85,B 0,C 180,E1 -9959.239,E2 -9959.239} C_VEL
LIN {X 0,Y 425.346,Z 229.001,A -85,B 0,C 180,E1 -9962.442,E2 -9962.442} C_VEL
LIN {X 0,Y 425.347,Z 229.004,A -85,B 0,C 180,E1 -9965.602,E2 -9965.602} C_VEL
LIN {X 0,Y 425.289,Z 229.009,A -85,B 0,C 180,E1 -9968.681,E2 -9968.681} C_VEL
LIN {X 0,Y 425.33,Z 229.006,A -85,B 0,C 180,E1 -9971.703,E2 -9971.703} C_VEL
LIN {X 0,Y 425.346,Z 229.004,A -85,B 0,C 180,E1 -9974.671,E2 -9974.671} C_VEL
LIN {X 0,Y 425.408,Z 228.997,A -85,B 0,C 180,E1 -9977.598,E2 -9977.598} C_VEL
LIN {X 0,Y 425.439,Z 228.993,A -85,B 0,C 180,E1 -9981.45,E2 -9981.45} C_VEL
LIN {X 0,Y 425.552,Z 228.978,A -85,B 0,C 180,E1 -9984.313,E2 -9984.313} C_VEL
LIN {X 0,Y 425.572,Z 228.975,A -85,B 0,C 180,E1 -9988.107,E2 -9988.107} C_VEL
LIN {X 0,Y 425.7,Z 228.96,A -85,B 0,C 180,E1 -9990,E2 -9990} C_VEL
LIN {X 0,Y 425.554,Z 228.978,A -85,B 0,C 180,E1 -9992.84,E2 -9992.84} C_VEL
LIN {X 0,Y 425.528,Z 228.982,A -85,B 0,C 180,E1 -9996.639,E2 -9996.639} C_VEL
LIN {X 0,Y 425.399,Z 228.996,A -85,B 0,C 180,E1 -9999.151,E2 -9999.151} C_VEL
LIN {X 0,Y 424.727,Z 229.081,A -85,B 0,C 180,E1 -9999.941,E2 -9999.941} C_VEL
LIN {X 0,Y 421.879,Z 229.437,A -85,B 0,C 180,E1 -10001.224,E2 -10001.224} C_VEL
LIN {X 0,Y 419.463,Z 229.738,A -85,B 0,C 180,E1 -10002.26,E2 -10002.26} C_VEL
LIN {X 0,Y 418.412,Z 229.868,A -85,B 0,C 180,E1 -10003.061,E2 -10003.061} C_VEL
LIN {X 0,Y 418.319,Z 229.878,A -85,B 0,C 180,E1 -10003.333,E2 -10003.333} C_VEL
LIN {X 0,Y 418.309,Z 229.881,A -85,B 0,C 180,E1 -10006.736,E2 -10006.736} C_VEL
LIN {X 0,Y 418.267,Z 229.884,A -85,B 0,C 180,E1 -10009.791,E2 -10009.791} C_VEL
LIN {X 0,Y 418.234,Z 229.891,A -85,B 0,C 180,E1 -10012.736,E2 -10012.736} C_VEL
LIN {X 0,Y 418.267,Z 229.885,A -85,B 0,C 180,E1 -10015.904,E2 -10015.904} C_VEL
LIN {X 0,Y 418.261,Z 229.867,A -85,B 0,C 180,E1 -10019.162,E2 -10019.162} C_VEL
LIN {X 0,Y 418.254,Z 229.879,A -85,B 0,C 180,E1 -10022.844,E2 -10022.844} C_VEL
LIN {X 0,Y 418.245,Z 229.877,A -85,B 0,C 180,E1 -10026.239,E2 -10026.239} C_VEL
LIN {X 0,Y 418.26,Z 229.879,A -85,B 0,C 180,E1 -10029.681,E2 -10029.681} C_VEL
LIN {X 0,Y 418.241,Z 229.857,A -85,B 0,C 180,E1 -10032.324,E2 -10032.324} C_VEL
LIN {X 0,Y 418.255,Z 229.879,A -85,B 0,C 180,E1 -10035.112,E2 -10035.112} C_VEL
LIN {X 0,Y 418.288,Z 229.882,A -85,B 0,C 180,E1 -10037.774,E2 -10037.774} C_VEL
LIN {X 0,Y 418.261,Z 229.883,A -85,B 0,C 180,E1 -10041.56,E2 -10041.56} C_VEL
LIN {X 0,Y 418.256,Z 229.874,A -85,B 0,C 180,E1 -10045.159,E2 -10045.159} C_VEL
LIN {X 0,Y 418.242,Z 229.882,A -85,B 0,C 180,E1 -10047.472,E2 -10047.472} C_VEL
LIN {X 0,Y 418.266,Z 229.877,A -85,B 0,C 180,E1 -10050.896,E2 -10050.896} C_VEL
LIN {X 0,Y 418.265,Z 229.878,A -85,B 0,C 180,E1 -10054.096,E2 -10054.096} C_VEL
LIN {X 0,Y 418.229,Z 229.888,A -85,B 0,C 180,E1 -10057.264,E2 -10057.264} C_VEL
LIN {X 0,Y 418.281,Z 229.861,A -85,B 0,C 180,E1 -10060.365,E2 -10060.365} C_VEL
LIN {X 0,Y 418.315,Z 229.872,A -85,B 0,C 180,E1 -10063.405,E2 -10063.405} C_VEL
LIN {X 0,Y 418.345,Z 229.872,A -85,B 0,C 180,E1 -10067,E2 -10067} C_VEL
LIN {X 0,Y 418.34,Z 229.85,A -85,B 0,C 180,E1 -10070.329,E2 -10070.329} C_VEL
LIN {X 0,Y 418.486,Z 229.853,A -85,B 0,C 180,E1 -10073.249,E2 -10073.249} C_VEL
LIN {X 0,Y 418.337,Z 229.878,A -85,B 0,C 180,E1 -10075.182,E2 -10075.182} C_VEL
LIN {X 0,Y 418.543,Z 229.834,A -85,B 0,C 180,E1 -10078.076,E2 -10078.076} C_VEL
LIN {X 0,Y 418.67,Z 229.81,A -85,B 0,C 180,E1 -10080.001,E2 -10080.001} C_VEL
LIN {X 0,Y 418.501,Z 229.849,A -85,B 0,C 180,E1 -10082.888,E2 -10082.888} C_VEL
LIN {X 0,Y 418.499,Z 229.85,A -85,B 0,C 180,E1 -10085.783,E2 -10085.783} C_VEL
LIN {X 0,Y 418.377,Z 229.852,A -85,B 0,C 180,E1 -10088.696,E2 -10088.696} C_VEL
LIN {X 0,Y 418.315,Z 229.868,A -85,B 0,C 180,E1 -10091.632,E2 -10091.632} C_VEL
LIN {X 0,Y 418.302,Z 229.878,A -85,B 0,C 180,E1 -10094.598,E2 -10094.598} C_VEL
LIN {X 0,Y 418.28,Z 229.863,A -85,B 0,C 180,E1 -10097.605,E2 -10097.605} C_VEL
LIN {X 0,Y 418.25,Z 229.876,A -85,B 0,C 180,E1 -10100.663,E2 -10100.663} C_VEL
LIN {X 0,Y 418.277,Z 229.878,A -85,B 0,C 180,E1 -10103.782,E2 -10103.782} C_VEL
LIN {X 0,Y 418.311,Z 229.863,A -85,B 0,C 180,E1 -10107.071,E2 -10107.071} C_VEL
LIN {X 0,Y 418.245,Z 229.886,A -85,B 0,C 180,E1 -10110.273,E2 -10110.273} C_VEL
LIN {X 0,Y 418.233,Z 229.875,A -85,B 0,C 180,E1 -10113.679,E2 -10113.679} C_VEL
LIN {X 0,Y 418.24,Z 229.885,A -85,B 0,C 180,E1 -10117.225,E2 -10117.225} C_VEL
LIN {X 0,Y 418.245,Z 229.878,A -85,B 0,C 180,E1 -10119.683,E2 -10119.683} C_VEL
LIN {X 0,Y 418.231,Z 229.891,A -85,B 0,C 180,E1 -10122.322,E2 -10122.322} C_VEL
LIN {X 0,Y 418.237,Z 229.884,A -85,B 0,C 180,E1 -10125.109,E2 -10125.109} C_VEL
LIN {X 0,Y 418.241,Z 229.886,A -85,B 0,C 180,E1 -10127.767,E2 -10127.767} C_VEL
LIN {X 0,Y 418.257,Z 229.875,A -85,B 0,C 180,E1 -10130.619,E2 -10130.619} C_VEL
LIN {X 0,Y 418.245,Z 229.878,A -85,B 0,C 180,E1 -10133.976,E2 -10133.976} C_VEL
LIN {X 0,Y 418.26,Z 229.88,A -85,B 0,C 180,E1 -10137.156,E2 -10137.156} C_VEL
LIN {X 0,Y 418.306,Z 230.064,A -85,B 0,C 180,E1 -10140.841,E2 -10140.841} C_VEL
LIN {X 0,Y 419.883,Z 238.039,A -85,B 0,C 180,E1 -10143.133,E2 -10143.133} C_VEL
LIN {X 0,Y 420.665,Z 244.541,A -85,B 0,C 180,E1 -10144.894,E2 -10144.894} C_VEL
LIN {X 0,Y 419.751,Z 258.611,A -85,B 0,C 180,E1 -10148.386,E2 -10148.386} C_VEL
LIN {X 0,Y 419.082,Z 268.523,A -85,B 0,C 180,E1 -10150.881,E2 -10150.881} C_VEL
LIN {X 0,Y 419.627,Z 271.938,A -85,B 0,C 180,E1 -10151.022,E2 -10151.022} C_VEL
LIN {X 0,Y 423.701,Z 294.757,A -85,B 0,C 180,E1 -10151.608,E2 -10151.608} C_VEL
LIN {X 0,Y 422.852,Z 373.44,A -85,B 0,C 180,E1 -10152.966,E2 -10152.966} C_VEL
LIN {X 0,Y 422.575,Z 383.337,A -85,B 0,C 180,E1 -10153.235,E2 -10153.235} C_VEL
LIN {X 0,Y 422.146,Z 393.314,A -85,B 0,C 180,E1 -10153.622,E2 -10153.622} C_VEL
LIN {X 0,Y 421.628,Z 402.669,A -85,B 0,C 180,E1 -10154.098,E2 -10154.098} C_VEL
LIN {X 0,Y 421.031,Z 412.812,A -85,B 0,C 180,E1 -10154.758,E2 -10154.758} C_VEL
LIN {X 0,Y 420.4,Z 421.808,A -85,B 0,C 180,E1 -10155.478,E2 -10155.478} C_VEL
LIN {X 0,Y 419.867,Z 429.803,A -85,B 0,C 180,E1 -10156.244,E2 -10156.244} C_VEL
LIN {X 0,Y 419.306,Z 437.936,A -85,B 0,C 180,E1 -10157.169,E2 -10157.169} C_VEL
LIN {X 0,Y 418.75,Z 445.155,A -85,B 0,C 180,E1 -10158.136,E2 -10158.136} C_VEL
LIN {X 0,Y 418.288,Z 451.357,A -85,B 0,C 180,E1 -10159.104,E2 -10159.104} C_VEL
LIN {X 0,Y 417.839,Z 457.895,A -85,B 0,C 180,E1 -10160.317,E2 -10160.317} C_VEL
LIN {X 0,Y 417.573,Z 462.397,A -85,B 0,C 180,E1 -10161.288,E2 -10161.288} C_VEL
LIN {X 0,Y 417.266,Z 467.888,A -85,B 0,C 180,E1 -10162.743,E2 -10162.743} C_VEL
LIN {X 0,Y 417.107,Z 472.211,A -85,B 0,C 180,E1 -10164.198,E2 -10164.198} C_VEL
LIN {X 0,Y 417.107,Z 474.579,A -85,B 0,C 180,E1 -10165.167,E2 -10165.167} C_VEL
LIN {X 0,Y 417.028,Z 477.761,A -85,B 0,C 180,E1 -10167.102,E2 -10167.102} C_VEL
LIN {X 0,Y 417.057,Z 478.819,A -85,B 0,C 180,E1 -10168.069,E2 -10168.069} C_VEL
LIN {X 0,Y 417.011,Z 479.406,A -85,B 0,C 180,E1 -10169.034,E2 -10169.034} C_VEL
LIN {X 0,Y 417.011,Z 479.406,A -85,B 0,C 180,E1 -10170.966,E2 -10170.966} C_VEL
LIN {X 0,Y 417.057,Z 478.819,A -85,B 0,C 180,E1 -10171.931,E2 -10171.931} C_VEL
LIN {X 0,Y 417.015,Z 476.375,A -85,B 0,C 180,E1 -10173.865,E2 -10173.865} C_VEL
LIN {X 0,Y 417.12,Z 473.429,A -85,B 0,C 180,E1 -10175.317,E2 -10175.317} C_VEL
LIN {X 0,Y 417.232,Z 469.442,A -85,B 0,C 180,E1 -10176.771,E2 -10176.771} C_VEL
LIN {X 0,Y 417.459,Z 464.313,A -85,B 0,C 180,E1 -10178.227,E2 -10178.227} C_VEL
LIN {X 0,Y 417.775,Z 459.051,A -85,B 0,C 180,E1 -10179.44,E2 -10179.44} C_VEL
LIN {X 0,Y 418.169,Z 452.733,A -85,B 0,C 180,E1 -10180.654,E2 -10180.654} C_VEL
LIN {X 0,Y 418.616,Z 446.782,A -85,B 0,C 180,E1 -10181.623,E2 -10181.623} C_VEL
LIN {X 0,Y 419.152,Z 439.855,A -85,B 0,C 180,E1 -10182.59,E2 -10182.59} C_VEL
LIN {X 0,Y 419.72,Z 431.673,A -85,B 0,C 180,E1 -10183.558,E2 -10183.558} C_VEL
LIN {X 0,Y 420.299,Z 423.022,A -85,B 0,C 180,E1 -10184.415,E2 -10184.415} C_VEL
LIN {X 0,Y 420.926,Z 414.444,A -85,B 0,C 180,E1 -10185.122,E2 -10185.122} C_VEL
LIN {X 0,Y 421.512,Z 404.683,A -85,B 0,C 180,E1 -10185.782,E2 -10185.782} C_VEL
LIN {X 0,Y 422.055,Z 394.601,A -85,B 0,C 180,E1 -10186.32,E2 -10186.32} C_VEL
LIN {X 0,Y 422.535,Z 385.087,A -85,B 0,C 180,E1 -10186.705,E2 -10186.705} C_VEL
LIN {X 0,Y 422.884,Z 374.774,A -85,B 0,C 180,E1 -10187.001,E2 -10187.001} C_VEL
LIN {X 0,Y 423.702,Z 299.528,A -85,B 0,C 180,E1 -10188.308,E2 -10188.308} C_VEL
LIN {X 0,Y 423.526,Z 293.51,A -85,B 0,C 180,E1 -10188.421,E2 -10188.421} C_VEL
LIN {X 0,Y 419.089,Z 268.793,A -85,B 0,C 180,E1 -10189.087,E2 -10189.087} C_VEL
LIN {X 0,Y 419.125,Z 267.49,A -85,B 0,C 180,E1 -10189.34,E2 -10189.34} C_VEL
LIN {X 0,Y 420.024,Z 254.697,A -85,B 0,C 180,E1 -10192.634,E2 -10192.634} C_VEL
LIN {X 0,Y 420.758,Z 244.833,A -85,B 0,C 180,E1 -10195.116,E2 -10195.116} C_VEL
LIN {X 0,Y 419.921,Z 238.178,A -85,B 0,C 180,E1 -10196.865,E2 -10196.865} C_VEL
LIN {X 0,Y 418.273,Z 229.918,A -85,B 0,C 180,E1 -10199.23,E2 -10199.23} C_VEL
LIN {X 0,Y 418.26,Z 229.881,A -85,B 0,C 180,E1 -10202.844,E2 -10202.844} C_VEL
LIN {X 0,Y 418.247,Z 229.879,A -85,B 0,C 180,E1 -10206.238,E2 -10206.238} C_VEL
LIN {X 0,Y 418.253,Z 229.872,A -85,B 0,C 180,E1 -10209.682,E2 -10209.682} C_VEL
LIN {X 0,Y 418.231,Z 229.886,A -85,B 0,C 180,E1 -10212.321,E2 -10212.321} C_VEL
LIN {X 0,Y 418.237,Z 229.884,A -85,B 0,C 180,E1 -10215.108,E2 -10215.108} C_VEL
LIN {X 0,Y 418.241,Z 229.889,A -85,B 0,C 180,E1 -10217.766,E2 -10217.766} C_VEL
LIN {X 0,Y 418.246,Z 229.877,A -85,B 0,C 180,E1 -10220.62,E2 -10220.62} C_VEL
LIN {X 0,Y 418.243,Z 229.882,A -85,B 0,C 180,E1 -10223.975,E2 -10223.975} C_VEL
LIN {X 0,Y 418.243,Z 229.881,A -85,B 0,C 180,E1 -10227.471,E2 -10227.471} C_VEL
LIN {X 0,Y 418.269,Z 229.881,A -85,B 0,C 180,E1 -10230.895,E2 -10230.895} C_VEL
LIN {X 0,Y 418.27,Z 229.871,A -85,B 0,C 180,E1 -10234.095,E2 -10234.095} C_VEL
LIN {X 0,Y 418.233,Z 229.89,A -85,B 0,C 180,E1 -10237.263,E2 -10237.263} C_VEL
LIN {X 0,Y 418.283,Z 229.866,A -85,B 0,C 180,E1 -10240.364,E2 -10240.364} C_VEL
LIN {X 0,Y 418.316,Z 229.871,A -85,B 0,C 180,E1 -10243.404,E2 -10243.404} C_VEL
LIN {X 0,Y 418.346,Z 229.872,A -85,B 0,C 180,E1 -10246.999,E2 -10246.999} C_VEL
LIN {X 0,Y 418.338,Z 229.851,A -85,B 0,C 180,E1 -10250.328,E2 -10250.328} C_VEL
LIN {X 0,Y 418.46,Z 229.858,A -85,B 0,C 180,E1 -10253.248,E2 -10253.248} C_VEL
LIN {X 0,Y 418.336,Z 229.876,A -85,B 0,C 180,E1 -10255.181,E2 -10255.181} C_VEL
LIN {X 0,Y 418.542,Z 229.84,A -85,B 0,C 180,E1 -10258.075,E2 -10258.075} C_VEL
LIN {X 0,Y 418.67,Z 229.81,A -85,B 0,C 180,E1 -10259.999,E2 -10259.999} C_VEL
LIN {X 0,Y 418.508,Z 229.849,A -85,B 0,C 180,E1 -10262.887,E2 -10262.887} C_VEL
LIN {X 0,Y 418.486,Z 229.853,A -85,B 0,C 180,E1 -10266.751,E2 -10266.751} C_VEL
LIN {X 0,Y 418.34,Z 229.85,A -85,B 0,C 180,E1 -10269.671,E2 -10269.671} C_VEL
LIN {X 0,Y 418.345,Z 229.872,A -85,B 0,C 180,E1 -10273,E2 -10273} C_VEL
LIN {X 0,Y 418.311,Z 229.871,A -85,B 0,C 180,E1 -10276.735,E2 -10276.735} C_VEL
LIN {X 0,Y 418.268,Z 229.863,A -85,B 0,C 180,E1 -10279.79,E2 -10279.79} C_VEL
LIN {X 0,Y 418.229,Z 229.888,A -85,B 0,C 180,E1 -10282.736,E2 -10282.736} C_VEL
LIN {X 0,Y 418.265,Z 229.878,A -85,B 0,C 180,E1 -10285.904,E2 -10285.904} C_VEL
LIN {X 0,Y 418.262,Z 229.878,A -85,B 0,C 180,E1 -10289.161,E2 -10289.161} C_VEL
LIN {X 0,Y 418.254,Z 229.879,A -85,B 0,C 180,E1 -10292.844,E2 -10292.844} C_VEL
LIN {X 0,Y 418.245,Z 229.885,A -85,B 0,C 180,E1 -10296.238,E2 -10296.238} C_VEL
LIN {X 0,Y 418.252,Z 229.883,A -85,B 0,C 180,E1 -10299.681,E2 -10299.681} C_VEL
LIN {X 0,Y 418.278,Z 229.883,A -85,B 0,C 180,E1 -10302.329,E2 -10302.329} C_VEL
LIN {X 0,Y 418.247,Z 229.88,A -85,B 0,C 180,E1 -10305.111,E2 -10305.111} C_VEL
LIN {X 0,Y 418.252,Z 229.855,A -85,B 0,C 180,E1 -10307.769,E2 -10307.769} C_VEL
LIN {X 0,Y 418.263,Z 229.88,A -85,B 0,C 180,E1 -10310.617,E2 -10310.617} C_VEL
LIN {X 0,Y 418.242,Z 229.875,A -85,B 0,C 180,E1 -10313.976,E2 -10313.976} C_VEL
LIN {X 0,Y 418.254,Z 229.879,A -85,B 0,C 180,E1 -10317.156,E2 -10317.156} C_VEL
LIN {X 0,Y 418.265,Z 229.868,A -85,B 0,C 180,E1 -10320.895,E2 -10320.895} C_VEL
LIN {X 0,Y 418.267,Z 229.885,A -85,B 0,C 180,E1 -10324.096,E2 -10324.096} C_VEL
LIN {X 0,Y 418.234,Z 229.891,A -85,B 0,C 180,E1 -10327.264,E2 -10327.264} C_VEL
LIN {X 0,Y 418.28,Z 229.883,A -85,B 0,C 180,E1 -10330.364,E2 -10330.364} C_VEL
LIN {X 0,Y 418.313,Z 229.881,A -85,B 0,C 180,E1 -10333.405,E2 -10333.405} C_VEL
LIN {X 0,Y 418.342,Z 229.877,A -85,B 0,C 180,E1 -10336.999,E2 -10336.999} C_VEL
LIN {X 0,Y 418.338,Z 229.876,A -85,B 0,C 180,E1 -10340.329,E2 -10340.329} C_VEL
LIN {X 0,Y 418.491,Z 229.858,A -85,B 0,C 180,E1 -10343.249,E2 -10343.249} C_VEL
LIN {X 0,Y 418.338,Z 229.878,A -85,B 0,C 180,E1 -10345.182,E2 -10345.182} C_VEL
LIN {X 0,Y 418.542,Z 229.851,A -85,B 0,C 180,E1 -10348.075,E2 -10348.075} C_VEL
LIN {X 0,Y 418.669,Z 229.836,A -85,B 0,C 180,E1 -10350,E2 -10350} C_VEL
LIN {X 0,Y 418.507,Z 229.856,A -85,B 0,C 180,E1 -10352.888,E2 -10352.888} C_VEL
LIN {X 0,Y 418.491,Z 229.858,A -85,B 0,C 180,E1 -10356.751,E2 -10356.751} C_VEL
LIN {X 0,Y 418.338,Z 229.876,A -85,B 0,C 180,E1 -10359.671,E2 -10359.671} C_VEL
LIN {X 0,Y 418.319,Z 229.878,A -85,B 0,C 180,E1 -10363.333,E2 -10363.333} C_VEL
LIN {X 0,Y 417.626,Z 229.966,A -85,B 0,C 180,E1 -10364.136,E2 -10364.136} C_VEL
LIN {X 0,Y 414.748,Z 230.324,A -85,B 0,C 180,E1 -10365.441,E2 -10365.441} C_VEL
LIN {X 0,Y 412.334,Z 230.626,A -85,B 0,C 180,E1 -10366.495,E2 -10366.495} C_VEL
LIN {X 0,Y 411.313,Z 230.752,A -85,B 0,C 180,E1 -10367.311,E2 -10367.311} C_VEL
LIN {X 0,Y 411.236,Z 230.76,A -85,B 0,C 180,E1 -10367.586,E2 -10367.586} C_VEL
LIN {X 0,Y 411.193,Z 230.767,A -85,B 0,C 180,E1 -10371.034,E2 -10371.034} C_VEL
LIN {X 0,Y 411.223,Z 230.764,A -85,B 0,C 180,E1 -10374.215,E2 -10374.215} C_VEL
LIN {X 0,Y 411.255,Z 230.757,A -85,B 0,C 180,E1 -10377.478,E2 -10377.478} C_VEL
LIN {X 0,Y 411.186,Z 230.765,A -85,B 0,C 180,E1 -10380.848,E2 -10380.848} C_VEL
LIN {X 0,Y 411.202,Z 230.744,A -85,B 0,C 180,E1 -10384.334,E2 -10384.334} C_VEL
LIN {X 0,Y 411.2,Z 230.766,A -85,B 0,C 180,E1 -10387.973,E2 -10387.973} C_VEL
LIN {X 0,Y 411.196,Z 230.738,A -85,B 0,C 180,E1 -10391.234,E2 -10391.234} C_VEL
LIN {X 0,Y 411.181,Z 230.758,A -85,B 0,C 180,E1 -10394.49,E2 -10394.49} C_VEL
LIN {X 0,Y 411.229,Z 230.758,A -85,B 0,C 180,E1 -10397.297,E2 -10397.297} C_VEL
LIN {X 0,Y 411.226,Z 230.757,A -85,B 0,C 180,E1 -10400.778,E2 -10400.778} C_VEL
LIN {X 0,Y 411.196,Z 230.754,A -85,B 0,C 180,E1 -10404.472,E2 -10404.472} C_VEL
LIN {X 0,Y 411.204,Z 230.756,A -85,B 0,C 180,E1 -10406.874,E2 -10406.874} C_VEL
LIN {X 0,Y 411.23,Z 230.754,A -85,B 0,C 180,E1 -10410.645,E2 -10410.645} C_VEL
LIN {X 0,Y 411.234,Z 230.745,A -85,B 0,C 180,E1 -10413.62,E2 -10413.62} C_VEL
LIN {X 0,Y 411.193,Z 230.762,A -85,B 0,C 180,E1 -10416.853,E2 -10416.853} C_VEL
LIN {X 0,Y 411.212,Z 230.743,A -85,B 0,C 180,E1 -10420.051,E2 -10420.051} C_VEL
LIN {X 0,Y 411.261,Z 230.747,A -85,B 0,C 180,E1 -10423.132,E2 -10423.132} C_VEL
LIN {X 0,Y 411.304,Z 230.748,A -85,B 0,C 180,E1 -10426.896,E2 -10426.896} C_VEL
LIN {X 0,Y 411.292,Z 230.728,A -85,B 0,C 180,E1 -10430.162,E2 -10430.162} C_VEL
LIN {X 0,Y 411.45,Z 230.728,A -85,B 0,C 180,E1 -10433.133,E2 -10433.133} C_VEL
LIN {X 0,Y 411.308,Z 230.752,A -85,B 0,C 180,E1 -10435.1,E2 -10435.1} C_VEL
LIN {X 0,Y 411.512,Z 230.71,A -85,B 0,C 180,E1 -10438.043,E2 -10438.043} C_VEL
LIN {X 0,Y 411.639,Z 230.685,A -85,B 0,C 180,E1 -10440.001,E2 -10440.001} C_VEL
LIN {X 0,Y 411.458,Z 230.727,A -85,B 0,C 180,E1 -10442.938,E2 -10442.938} C_VEL
LIN {X 0,Y 411.424,Z 230.732,A -85,B 0,C 180,E1 -10446.868,E2 -10446.868} C_VEL
LIN {X 0,Y 411.291,Z 230.728,A -85,B 0,C 180,E1 -10449.839,E2 -10449.839} C_VEL
LIN {X 0,Y 411.305,Z 230.751,A -85,B 0,C 180,E1 -10453.105,E2 -10453.105} C_VEL
LIN {X 0,Y 411.257,Z 230.744,A -85,B 0,C 180,E1 -10456.889,E2 -10456.889} C_VEL
LIN {X 0,Y 411.231,Z 230.744,A -85,B 0,C 180,E1 -10459.987,E2 -10459.987} C_VEL
LIN {X 0,Y 411.197,Z 230.762,A -85,B 0,C 180,E1 -10463.148,E2 -10463.148} C_VEL
LIN {X 0,Y 411.238,Z 230.745,A -85,B 0,C 180,E1 -10466.381,E2 -10466.381} C_VEL
LIN {X 0,Y 411.201,Z 230.76,A -85,B 0,C 180,E1 -10469.713,E2 -10469.713} C_VEL
LIN {X 0,Y 411.205,Z 230.751,A -85,B 0,C 180,E1 -10473.157,E2 -10473.157} C_VEL
LIN {X 0,Y 411.193,Z 230.766,A -85,B 0,C 180,E1 -10476.553,E2 -10476.553} C_VEL
LIN {X 0,Y 411.21,Z 230.755,A -85,B 0,C 180,E1 -10479.728,E2 -10479.728} C_VEL
LIN {X 0,Y 411.175,Z 230.764,A -85,B 0,C 180,E1 -10483.134,E2 -10483.134} C_VEL
LIN {X 0,Y 411.17,Z 230.766,A -85,B 0,C 180,E1 -10485.881,E2 -10485.881} C_VEL
LIN {X 0,Y 411.165,Z 230.753,A -85,B 0,C 180,E1 -10488.772,E2 -10488.772} C_VEL
LIN {X 0,Y 411.208,Z 230.762,A -85,B 0,C 180,E1 -10491.832,E2 -10491.832} C_VEL
LIN {X 0,Y 411.213,Z 230.757,A -85,B 0,C 180,E1 -10495.122,E2 -10495.122} C_VEL
LIN {X 0,Y 411.168,Z 230.763,A -85,B 0,C 180,E1 -10498.003,E2 -10498.003} C_VEL
LIN {X 0,Y 411.262,Z 230.943,A -85,B 0,C 180,E1 -10500.574,E2 -10500.574} C_VEL
LIN {X 0,Y 413.151,Z 240.804,A -85,B 0,C 180,E1 -10503.479,E2 -10503.479} C_VEL
LIN {X 0,Y 413.691,Z 246.014,A -85,B 0,C 180,E1 -10504.868,E2 -10504.868} C_VEL
LIN {X 0,Y 412.692,Z 260.511,A -85,B 0,C 180,E1 -10508.523,E2 -10508.523} C_VEL
LIN {X 0,Y 412.147,Z 268.33,A -85,B 0,C 180,E1 -10510.547,E2 -10510.547} C_VEL
LIN {X 0,Y 412.701,Z 271.744,A -85,B 0,C 180,E1 -10510.691,E2 -10510.691} C_VEL
LIN {X 0,Y 416.972,Z 295.806,A -85,B 0,C 180,E1 -10511.323,E2 -10511.323} C_VEL
LIN {X 0,Y 416.078,Z 373.248,A -85,B 0,C 180,E1 -10512.68,E2 -10512.68} C_VEL
LIN {X 0,Y 415.793,Z 383.145,A -85,B 0,C 180,E1 -10512.953,E2 -10512.953} C_VEL
LIN {X 0,Y 415.346,Z 393.121,A -85,B 0,C 180,E1 -10513.346,E2 -10513.346} C_VEL
LIN {X 0,Y 414.792,Z 402.476,A -85,B 0,C 180,E1 -10513.829,E2 -10513.829} C_VEL
LIN {X 0,Y 414.158,Z 412.618,A -85,B 0,C 180,E1 -10514.498,E2 -10514.498} C_VEL
LIN {X 0,Y 413.502,Z 421.615,A -85,B 0,C 180,E1 -10515.23,E2 -10515.23} C_VEL
LIN {X 0,Y 412.895,Z 430.124,A -85,B 0,C 180,E1 -10516.064,E2 -10516.064} C_VEL
LIN {X 0,Y 412.347,Z 437.742,A -85,B 0,C 180,E1 -10516.948,E2 -10516.948} C_VEL
LIN {X 0,Y 411.769,Z 444.961,A -85,B 0,C 180,E1 -10517.932,E2 -10517.932} C_VEL
LIN {X 0,Y 411.295,Z 451.164,A -85,B 0,C 180,E1 -10518.917,E2 -10518.917} C_VEL
LIN {X 0,Y 410.817,Z 457.702,A -85,B 0,C 180,E1 -10520.15,E2 -10520.15} C_VEL
LIN {X 0,Y 410.532,Z 462.204,A -85,B 0,C 180,E1 -10521.137,E2 -10521.137} C_VEL
LIN {X 0,Y 410.186,Z 467.694,A -85,B 0,C 180,E1 -10522.617,E2 -10522.617} C_VEL
LIN {X 0,Y 410.013,Z 472.018,A -85,B 0,C 180,E1 -10524.097,E2 -10524.097} C_VEL
LIN {X 0,Y 410.019,Z 474.386,A -85,B 0,C 180,E1 -10525.084,E2 -10525.084} C_VEL
LIN {X 0,Y 409.933,Z 476.182,A -85,B 0,C 180,E1 -10526.068,E2 -10526.068} C_VEL
LIN {X 0,Y 409.967,Z 478.627,A -85,B 0,C 180,E1 -10528.035,E2 -10528.035} C_VEL
LIN {X 0,Y 409.936,Z 479.214,A -85,B 0,C 180,E1 -10529.018,E2 -10529.018} C_VEL
LIN {X 0,Y 409.936,Z 479.214,A -85,B 0,C 180,E1 -10530.982,E2 -10530.982} C_VEL
LIN {X 0,Y 409.967,Z 478.627,A -85,B 0,C 180,E1 -10531.965,E2 -10531.965} C_VEL
LIN {X 0,Y 409.933,Z 476.182,A -85,B 0,C 180,E1 -10533.932,E2 -10533.932} C_VEL
LIN {X 0,Y 410.016,Z 473.235,A -85,B 0,C 180,E1 -10535.41,E2 -10535.41} C_VEL
LIN {X 0,Y 410.164,Z 469.249,A -85,B 0,C 180,E1 -10536.889,E2 -10536.889} C_VEL
LIN {X 0,Y 410.414,Z 464.12,A -85,B 0,C 180,E1 -10538.369,E2 -10538.369} C_VEL
LIN {X 0,Y 410.747,Z 458.858,A -85,B 0,C 180,E1 -10539.603,E2 -10539.603} C_VEL
LIN {X 0,Y 411.153,Z 452.539,A -85,B 0,C 180,E1 -10540.838,E2 -10540.838} C_VEL
LIN {X 0,Y 411.635,Z 446.588,A -85,B 0,C 180,E1 -10541.822,E2 -10541.822} C_VEL
LIN {X 0,Y 412.189,Z 439.661,A -85,B 0,C 180,E1 -10542.806,E2 -10542.806} C_VEL
LIN {X 0,Y 412.795,Z 431.48,A -85,B 0,C 180,E1 -10543.789,E2 -10543.789} C_VEL
LIN {X 0,Y 413.405,Z 422.951,A -85,B 0,C 180,E1 -10544.649,E2 -10544.649} C_VEL
LIN {X 0,Y 414.072,Z 414.251,A -85,B 0,C 180,E1 -10545.379,E2 -10545.379} C_VEL
LIN {X 0,Y 414.678,Z 404.491,A -85,B 0,C 180,E1 -10546.049,E2 -10546.049} C_VEL
LIN {X 0,Y 415.227,Z 394.407,A -85,B 0,C 180,E1 -10546.596,E2 -10546.596} C_VEL
LIN {X 0,Y 415.722,Z 384.894,A -85,B 0,C 180,E1 -10546.987,E2 -10546.987} C_VEL
LIN {X 0,Y 416.093,Z 374.581,A -85,B 0,C 180,E1 -10547.287,E2 -10547.287} C_VEL
LIN {X 0,Y 416.963,Z 299.335,A -85,B 0,C 180,E1 -10548.615,E2 -10548.615} C_VEL
LIN {X 0,Y 416.812,Z 294.637,A -85,B 0,C 180,E1 -10548.706,E2 -10548.706} C_VEL
LIN {X 0,Y 412.156,Z 268.602,A -85,B 0,C 180,E1 -10549.421,E2 -10549.421} C_VEL
LIN {X 0,Y 412.18,Z 267.299,A -85,B 0,C 180,E1 -10549.679,E2 -10549.679} C_VEL
LIN {X 0,Y 413.116,Z 254.522,A -85,B 0,C 180,E1 -10553.034,E2 -10553.034} C_VEL
LIN {X 0,Y 413.755,Z 245.125,A -85,B 0,C 180,E1 -10555.449,E2 -10555.449} C_VEL
LIN {X 0,Y 412.494,Z 237.112,A -85,B 0,C 180,E1 -10557.628,E2 -10557.628} C_VEL
LIN {X 0,Y 411.242,Z 230.813,A -85,B 0,C 180,E1 -10559.485,E2 -10559.485} C_VEL
LIN {X 0,Y 411.209,Z 230.761,A -85,B 0,C 180,E1 -10563.155,E2 -10563.155} C_VEL
LIN {X 0,Y 411.195,Z 230.761,A -85,B 0,C 180,E1 -10566.552,E2 -10566.552} C_VEL
LIN {X 0,Y 411.217,Z 230.747,A -85,B 0,C 180,E1 -10569.728,E2 -10569.728} C_VEL
LIN {X 0,Y 411.175,Z 230.765,A -85,B 0,C 180,E1 -10573.133,E2 -10573.133} C_VEL
LIN {X 0,Y 411.169,Z 230.765,A -85,B 0,C 180,E1 -10575.881,E2 -10575.881} C_VEL
LIN {X 0,Y 411.164,Z 230.764,A -85,B 0,C 180,E1 -10578.771,E2 -10578.771} C_VEL
LIN {X 0,Y 411.193,Z 230.765,A -85,B 0,C 180,E1 -10582.026,E2 -10582.026} C_VEL
LIN {X 0,Y 411.193,Z 230.752,A -85,B 0,C 180,E1 -10585.665,E2 -10585.665} C_VEL
LIN {X 0,Y 411.19,Z 230.766,A -85,B 0,C 180,E1 -10589.152,E2 -10589.152} C_VEL
LIN {X 0,Y 411.26,Z 230.742,A -85,B 0,C 180,E1 -10592.522,E2 -10592.522} C_VEL
LIN {X 0,Y 411.221,Z 230.759,A -85,B 0,C 180,E1 -10595.784,E2 -10595.784} C_VEL
LIN {X 0,Y 411.197,Z 230.76,A -85,B 0,C 180,E1 -10598.965,E2 -10598.965} C_VEL
LIN {X 0,Y 411.245,Z 230.739,A -85,B 0,C 180,E1 -10602.084,E2 -10602.084} C_VEL
LIN {X 0,Y 411.26,Z 230.757,A -85,B 0,C 180,E1 -10605.147,E2 -10605.147} C_VEL
LIN {X 0,Y 411.283,Z 230.743,A -85,B 0,C 180,E1 -10608.167,E2 -10608.167} C_VEL
LIN {X 0,Y 411.318,Z 230.729,A -85,B 0,C 180,E1 -10611.153,E2 -10611.153} C_VEL
LIN {X 0,Y 411.444,Z 230.729,A -85,B 0,C 180,E1 -10614.117,E2 -10614.117} C_VEL
LIN {X 0,Y 411.511,Z 230.716,A -85,B 0,C 180,E1 -10618.042,E2 -10618.042} C_VEL
LIN {X 0,Y 411.639,Z 230.685,A -85,B 0,C 180,E1 -10619.999,E2 -10619.999} C_VEL
LIN {X 0,Y 411.464,Z 230.726,A -85,B 0,C 180,E1 -10622.937,E2 -10622.937} C_VEL
LIN {X 0,Y 411.45,Z 230.728,A -85,B 0,C 180,E1 -10626.867,E2 -10626.867} C_VEL
LIN {X 0,Y 411.292,Z 230.728,A -85,B 0,C 180,E1 -10629.838,E2 -10629.838} C_VEL
LIN {X 0,Y 411.304,Z 230.748,A -85,B 0,C 180,E1 -10633.104,E2 -10633.104} C_VEL
LIN {X 0,Y 411.261,Z 230.747,A -85,B 0,C 180,E1 -10636.868,E2 -10636.868} C_VEL
LIN {X 0,Y 411.228,Z 230.741,A -85,B 0,C 180,E1 -10639.986,E2 -10639.986} C_VEL
LIN {X 0,Y 411.193,Z 230.762,A -85,B 0,C 180,E1 -10643.147,E2 -10643.147} C_VEL
LIN {X 0,Y 411.234,Z 230.745,A -85,B 0,C 180,E1 -10646.38,E2 -10646.38} C_VEL
LIN {X 0,Y 411.197,Z 230.759,A -85,B 0,C 180,E1 -10649.712,E2 -10649.712} C_VEL
LIN {X 0,Y 411.203,Z 230.756,A -85,B 0,C 180,E1 -10653.155,E2 -10653.155} C_VEL
LIN {X 0,Y 411.192,Z 230.765,A -85,B 0,C 180,E1 -10656.553,E2 -10656.553} C_VEL
LIN {X 0,Y 411.216,Z 230.758,A -85,B 0,C 180,E1 -10659.728,E2 -10659.728} C_VEL
LIN {X 0,Y 411.226,Z 230.758,A -85,B 0,C 180,E1 -10663.126,E2 -10663.126} C_VEL
LIN {X 0,Y 411.168,Z 230.752,A -85,B 0,C 180,E1 -10665.88,E2 -10665.88} C_VEL
LIN {X 0,Y 411.208,Z 230.743,A -85,B 0,C 180,E1 -10669.499,E2 -10669.499} C_VEL
LIN {X 0,Y 411.2,Z 230.766,A -85,B 0,C 180,E1 -10672.027,E2 -10672.027} C_VEL
LIN {X 0,Y 411.202,Z 230.744,A -85,B 0,C 180,E1 -10675.666,E2 -10675.666} C_VEL
LIN {X 0,Y 411.186,Z 230.765,A -85,B 0,C 180,E1 -10679.152,E2 -10679.152} C_VEL
LIN {X 0,Y 411.255,Z 230.757,A -85,B 0,C 180,E1 -10682.522,E2 -10682.522} C_VEL
LIN {X 0,Y 411.223,Z 230.764,A -85,B 0,C 180,E1 -10685.785,E2 -10685.785} C_VEL
LIN {X 0,Y 411.193,Z 230.767,A -85,B 0,C 180,E1 -10688.966,E2 -10688.966} C_VEL
LIN {X 0,Y 411.249,Z 230.76,A -85,B 0,C 180,E1 -10692.085,E2 -10692.085} C_VEL
LIN {X 0,Y 411.257,Z 230.76,A -85,B 0,C 180,E1 -10695.147,E2 -10695.147} C_VEL
LIN {X 0,Y 411.281,Z 230.756,A -85,B 0,C 180,E1 -10698.167,E2 -10698.167} C_VEL
LIN {X 0,Y 411.478,Z 230.732,A -85,B 0,C 180,E1 -10702.147,E2 -10702.147} C_VEL
LIN {X 0,Y 411.473,Z 230.732,A -85,B 0,C 180,E1 -10704.118,E2 -10704.118} C_VEL
LIN {X 0,Y 411.511,Z 230.727,A -85,B 0,C 180,E1 -10708.043,E2 -10708.043} C_VEL
LIN {X 0,Y 411.639,Z 230.712,A -85,B 0,C 180,E1 -10710,E2 -10710} C_VEL
LIN {X 0,Y 411.463,Z 230.734,A -85,B 0,C 180,E1 -10712.937,E2 -10712.937} C_VEL
LIN {X 0,Y 411.458,Z 230.735,A -85,B 0,C 180,E1 -10716.867,E2 -10716.867} C_VEL
LIN {X 0,Y 411.29,Z 230.754,A -85,B 0,C 180,E1 -10719.839,E2 -10719.839} C_VEL
LIN {X 0,Y 411.28,Z 230.756,A -85,B 0,C 180,E1 -10723.321,E2 -10723.321} C_VEL
LIN {X 0,Y 411.253,Z 230.761,A -85,B 0,C 180,E1 -10726.889,E2 -10726.889} C_VEL
LIN {X 0,Y 411.236,Z 230.76,A -85,B 0,C 180,E1 -10727.586,E2 -10727.586} C_VEL
LIN {X 0,Y 410.576,Z 230.845,A -85,B 0,C 180,E1 -10728.404,E2 -10728.404} C_VEL
LIN {X 0,Y 407.688,Z 231.202,A -85,B 0,C 180,E1 -10729.732,E2 -10729.732} C_VEL
LIN {X 0,Y 405.244,Z 231.509,A -85,B 0,C 180,E1 -10730.805,E2 -10730.805} C_VEL
LIN {X 0,Y 404.208,Z 231.635,A -85,B 0,C 180,E1 -10731.635,E2 -10731.635} C_VEL
LIN {X 0,Y 404.132,Z 231.644,A -85,B 0,C 180,E1 -10731.916,E2 -10731.916} C_VEL
LIN {X 0,Y 404.212,Z 231.635,A -85,B 0,C 180,E1 -10735.297,E2 -10735.297} C_VEL
LIN {X 0,Y 404.191,Z 231.633,A -85,B 0,C 180,E1 -10738,E2 -10738} C_VEL
LIN {X 0,Y 404.135,Z 231.643,A -85,B 0,C 180,E1 -10741.558,E2 -10741.558} C_VEL
LIN {X 0,Y 404.182,Z 231.618,A -85,B 0,C 180,E1 -10745.016,E2 -10745.016} C_VEL
LIN {X 0,Y 404.159,Z 231.638,A -85,B 0,C 180,E1 -10748.756,E2 -10748.756} C_VEL
LIN {X 0,Y 404.146,Z 231.611,A -85,B 0,C 180,E1 -10751.604,E2 -10751.604} C_VEL
LIN {X 0,Y 404.149,Z 231.633,A -85,B 0,C 180,E1 -10754.524,E2 -10754.524} C_VEL
LIN {X 0,Y 404.207,Z 231.633,A -85,B 0,C 180,E1 -10757.306,E2 -10757.306} C_VEL
LIN {X 0,Y 404.165,Z 231.632,A -85,B 0,C 180,E1 -10759.956,E2 -10759.956} C_VEL
LIN {X 0,Y 404.137,Z 231.642,A -85,B 0,C 180,E1 -10763.125,E2 -10763.125} C_VEL
LIN {X 0,Y 404.142,Z 231.634,A -85,B 0,C 180,E1 -10766.188,E2 -10766.188} C_VEL
LIN {X 0,Y 404.142,Z 231.645,A -85,B 0,C 180,E1 -10769.715,E2 -10769.715} C_VEL
LIN {X 0,Y 404.192,Z 231.617,A -85,B 0,C 180,E1 -10773.123,E2 -10773.123} C_VEL
LIN {X 0,Y 404.171,Z 231.635,A -85,B 0,C 180,E1 -10775.335,E2 -10775.335} C_VEL
LIN {X 0,Y 404.136,Z 231.636,A -85,B 0,C 180,E1 -10778.581,E2 -10778.581} C_VEL
LIN {X 0,Y 404.208,Z 231.618,A -85,B 0,C 180,E1 -10781.762,E2 -10781.762} C_VEL
LIN {X 0,Y 404.205,Z 231.633,A -85,B 0,C 180,E1 -10784.883,E2 -10784.883} C_VEL
LIN {X 0,Y 404.255,Z 231.617,A -85,B 0,C 180,E1 -10787.959,E2 -10787.959} C_VEL
LIN {X 0,Y 404.403,Z 231.601,A -85,B 0,C 180,E1 -10792.13,E2 -10792.13} C_VEL
LIN {X 0,Y 404.418,Z 231.606,A -85,B 0,C 180,E1 -10794.016,E2 -10794.016} C_VEL
LIN {X 0,Y 404.481,Z 231.586,A -85,B 0,C 180,E1 -10798.009,E2 -10798.009} C_VEL
LIN {X 0,Y 404.609,Z 231.56,A -85,B 0,C 180,E1 -10800.001,E2 -10800.001} C_VEL
LIN {X 0,Y 404.416,Z 231.604,A -85,B 0,C 180,E1 -10802.989,E2 -10802.989} C_VEL
LIN {X 0,Y 404.369,Z 231.608,A -85,B 0,C 180,E1 -10806.989,E2 -10806.989} C_VEL
LIN {X 0,Y 404.256,Z 231.604,A -85,B 0,C 180,E1 -10810.012,E2 -10810.012} C_VEL
LIN {X 0,Y 404.266,Z 231.627,A -85,B 0,C 180,E1 -10813.212,E2 -10813.212} C_VEL
LIN {X 0,Y 404.216,Z 231.619,A -85,B 0,C 180,E1 -10817.007,E2 -10817.007} C_VEL
LIN {X 0,Y 404.164,Z 231.626,A -85,B 0,C 180,E1 -10820.352,E2 -10820.352} C_VEL
LIN {X 0,Y 404.164,Z 231.636,A -85,B 0,C 180,E1 -10823.575,E2 -10823.575} C_VEL
LIN {X 0,Y 404.184,Z 231.625,A -85,B 0,C 180,E1 -10825.767,E2 -10825.767} C_VEL
LIN {X 0,Y 404.196,Z 231.622,A -85,B 0,C 180,E1 -10828,E2 -10828} C_VEL
LIN {X 0,Y 404.139,Z 231.64,A -85,B 0,C 180,E1 -10831.558,E2 -10831.558} C_VEL
LIN {X 0,Y 404.175,Z 231.632,A -85,B 0,C 180,E1 -10835.018,E2 -10835.018} C_VEL
LIN {X 0,Y 404.151,Z 231.636,A -85,B 0,C 180,E1 -10838.758,E2 -10838.758} C_VEL
LIN {X 0,Y 404.124,Z 231.642,A -85,B 0,C 180,E1 -10841.6,E2 -10841.6} C_VEL
LIN {X 0,Y 404.147,Z 231.638,A -85,B 0,C 180,E1 -10844.522,E2 -10844.522} C_VEL
LIN {X 0,Y 404.138,Z 231.641,A -85,B 0,C 180,E1 -10847.296,E2 -10847.296} C_VEL
LIN {X 0,Y 404.171,Z 231.621,A -85,B 0,C 180,E1 -10849.956,E2 -10849.956} C_VEL
LIN {X 0,Y 404.138,Z 231.64,A -85,B 0,C 180,E1 -10853.125,E2 -10853.125} C_VEL
LIN {X 0,Y 404.147,Z 231.645,A -85,B 0,C 180,E1 -10856.188,E2 -10856.188} C_VEL
LIN {X 0,Y 404.192,Z 231.633,A -85,B 0,C 180,E1 -10860.101,E2 -10860.101} C_VEL
LIN {X 0,Y 404.263,Z 232.003,A -85,B 0,C 180,E1 -10860.371,E2 -10860.371} C_VEL
LIN {X 0,Y 406.136,Z 241.668,A -85,B 0,C 180,E1 -10863.262,E2 -10863.262} C_VEL
LIN {X 0,Y 406.738,Z 246.88,A -85,B 0,C 180,E1 -10864.681,E2 -10864.681} C_VEL
LIN {X 0,Y 405.793,Z 260.328,A -85,B 0,C 180,E1 -10868.139,E2 -10868.139} C_VEL
LIN {X 0,Y 405.189,Z 268.164,A -85,B 0,C 180,E1 -10870.203,E2 -10870.203} C_VEL
LIN {X 0,Y 405.971,Z 272.425,A -85,B 0,C 180,E1 -10870.374,E2 -10870.374} C_VEL
LIN {X 0,Y 410.236,Z 296.538,A -85,B 0,C 180,E1 -10871.021,E2 -10871.021} C_VEL
LIN {X 0,Y 409.322,Z 373.055,A -85,B 0,C 180,E1 -10872.385,E2 -10872.385} C_VEL
LIN {X 0,Y 409.013,Z 382.952,A -85,B 0,C 180,E1 -10872.662,E2 -10872.662} C_VEL
LIN {X 0,Y 408.532,Z 392.928,A -85,B 0,C 180,E1 -10873.06,E2 -10873.06} C_VEL
LIN {X 0,Y 407.964,Z 402.283,A -85,B 0,C 180,E1 -10873.551,E2 -10873.551} C_VEL
LIN {X 0,Y 407.327,Z 412.425,A -85,B 0,C 180,E1 -10874.232,E2 -10874.232} C_VEL
LIN {X 0,Y 406.616,Z 421.421,A -85,B 0,C 180,E1 -10874.974,E2 -10874.974} C_VEL
LIN {X 0,Y 406.015,Z 429.531,A -85,B 0,C 180,E1 -10875.778,E2 -10875.778} C_VEL
LIN {X 0,Y 405.379,Z 437.547,A -85,B 0,C 180,E1 -10876.72,E2 -10876.72} C_VEL
LIN {X 0,Y 404.804,Z 444.768,A -85,B 0,C 180,E1 -10877.721,E2 -10877.721} C_VEL
LIN {X 0,Y 404.298,Z 450.97,A -85,B 0,C 180,E1 -10878.723,E2 -10878.723} C_VEL
LIN {X 0,Y 403.811,Z 457.508,A -85,B 0,C 180,E1 -10879.977,E2 -10879.977} C_VEL
LIN {X 0,Y 403.49,Z 462.01,A -85,B 0,C 180,E1 -10880.981,E2 -10880.981} C_VEL
LIN {X 0,Y 403.133,Z 467.501,A -85,B 0,C 180,E1 -10882.487,E2 -10882.487} C_VEL
LIN {X 0,Y 402.94,Z 471.825,A -85,B 0,C 180,E1 -10883.993,E2 -10883.993} C_VEL
LIN {X 0,Y 402.931,Z 474.192,A -85,B 0,C 180,E1 -10884.997,E2 -10884.997} C_VEL
LIN {X 0,Y 402.853,Z 475.989,A -85,B 0,C 180,E1 -10885.999,E2 -10885.999} C_VEL
LIN {X 0,Y 402.865,Z 478.434,A -85,B 0,C 180,E1 -10888.001,E2 -10888.001} C_VEL
LIN {X 0,Y 402.863,Z 479.022,A -85,B 0,C 180,E1 -10889,E2 -10889} C_VEL
LIN {X 0,Y 402.863,Z 479.022,A -85,B 0,C 180,E1 -10891,E2 -10891} C_VEL
LIN {X 0,Y 402.865,Z 478.434,A -85,B 0,C 180,E1 -10891.999,E2 -10891.999} C_VEL
LIN {X 0,Y 402.853,Z 475.989,A -85,B 0,C 180,E1 -10894.001,E2 -10894.001} C_VEL
LIN {X 0,Y 402.914,Z 473.042,A -85,B 0,C 180,E1 -10895.505,E2 -10895.505} C_VEL
LIN {X 0,Y 403.076,Z 469.055,A -85,B 0,C 180,E1 -10897.01,E2 -10897.01} C_VEL
LIN {X 0,Y 403.357,Z 463.926,A -85,B 0,C 180,E1 -10898.517,E2 -10898.517} C_VEL
LIN {X 0,Y 403.709,Z 458.664,A -85,B 0,C 180,E1 -10899.772,E2 -10899.772} C_VEL
LIN {X 0,Y 404.147,Z 452.345,A -85,B 0,C 180,E1 -10901.028,E2 -10901.028} C_VEL
LIN {X 0,Y 404.658,Z 446.395,A -85,B 0,C 180,E1 -10902.029,E2 -10902.029} C_VEL
LIN {X 0,Y 405.229,Z 439.467,A -85,B 0,C 180,E1 -10903.03,E2 -10903.03} C_VEL
LIN {X 0,Y 405.855,Z 431.286,A -85,B 0,C 180,E1 -10904.03,E2 -10904.03} C_VEL
LIN {X 0,Y 406.498,Z 422.908,A -85,B 0,C 180,E1 -10904.89,E2 -10904.89} C_VEL
LIN {X 0,Y 407.2,Z 414.057,A -85,B 0,C 180,E1 -10905.645,E2 -10905.645} C_VEL
LIN {X 0,Y 407.853,Z 404.298,A -85,B 0,C 180,E1 -10906.325,E2 -10906.325} C_VEL
LIN {X 0,Y 408.434,Z 394.215,A -85,B 0,C 180,E1 -10906.88,E2 -10906.88} C_VEL
LIN {X 0,Y 408.95,Z 384.701,A -85,B 0,C 180,E1 -10907.277,E2 -10907.277} C_VEL
LIN {X 0,Y 409.316,Z 374.388,A -85,B 0,C 180,E1 -10907.583,E2 -10907.583} C_VEL
LIN {X 0,Y 410.269,Z 297.54,A -85,B 0,C 180,E1 -10908.959,E2 -10908.959} C_VEL
LIN {X 0,Y 406.592,Z 275.792,A -85,B 0,C 180,E1 -10909.534,E2 -10909.534} C_VEL
LIN {X 0,Y 405.194,Z 268.346,A -85,B 0,C 180,E1 -10909.774,E2 -10909.774} C_VEL
LIN {X 0,Y 405.308,Z 266.158,A -85,B 0,C 180,E1 -10910.292,E2 -10910.292} C_VEL
LIN {X 0,Y 406.422,Z 252.322,A -85,B 0,C 180,E1 -10913.976,E2 -10913.976} C_VEL
LIN {X 0,Y 406.778,Z 246.178,A -85,B 0,C 180,E1 -10915.59,E2 -10915.59} C_VEL
LIN {X 0,Y 405.439,Z 237.886,A -85,B 0,C 180,E1 -10917.906,E2 -10917.906} C_VEL
LIN {X 0,Y 404.229,Z 231.7,A -85,B 0,C 180,E1 -10919.753,E2 -10919.753} C_VEL
LIN {X 0,Y 404.173,Z 231.639,A -85,B 0,C 180,E1 -10923.42,E2 -10923.42} C_VEL
LIN {X 0,Y 404.144,Z 231.635,A -85,B 0,C 180,E1 -10926.246,E2 -10926.246} C_VEL
LIN {X 0,Y 404.158,Z 231.637,A -85,B 0,C 180,E1 -10928.756,E2 -10928.756} C_VEL
LIN {X 0,Y 404.124,Z 231.632,A -85,B 0,C 180,E1 -10931.599,E2 -10931.599} C_VEL
LIN {X 0,Y 404.147,Z 231.638,A -85,B 0,C 180,E1 -10934.522,E2 -10934.522} C_VEL
LIN {X 0,Y 404.138,Z 231.643,A -85,B 0,C 180,E1 -10937.295,E2 -10937.295} C_VEL
LIN {X 0,Y 404.17,Z 231.631,A -85,B 0,C 180,E1 -10939.955,E2 -10939.955} C_VEL
LIN {X 0,Y 404.136,Z 231.644,A -85,B 0,C 180,E1 -10943.125,E2 -10943.125} C_VEL
LIN {X 0,Y 404.138,Z 231.631,A -85,B 0,C 180,E1 -10946.187,E2 -10946.187} C_VEL
LIN {X 0,Y 404.146,Z 231.642,A -85,B 0,C 180,E1 -10949.714,E2 -10949.714} C_VEL
LIN {X 0,Y 404.195,Z 231.619,A -85,B 0,C 180,E1 -10953.122,E2 -10953.122} C_VEL
LIN {X 0,Y 404.175,Z 231.634,A -85,B 0,C 180,E1 -10955.334,E2 -10955.334} C_VEL
LIN {X 0,Y 404.139,Z 231.639,A -85,B 0,C 180,E1 -10958.58,E2 -10958.58} C_VEL
LIN {X 0,Y 404.204,Z 231.615,A -85,B 0,C 180,E1 -10961.761,E2 -10961.761} C_VEL
LIN {X 0,Y 404.206,Z 231.632,A -85,B 0,C 180,E1 -10964.881,E2 -10964.881} C_VEL
LIN {X 0,Y 404.256,Z 231.619,A -85,B 0,C 180,E1 -10967.958,E2 -10967.958} C_VEL
LIN {X 0,Y 404.265,Z 231.605,A -85,B 0,C 180,E1 -10970.998,E2 -10970.998} C_VEL
LIN {X 0,Y 404.393,Z 231.607,A -85,B 0,C 180,E1 -10974.014,E2 -10974.014} C_VEL
LIN {X 0,Y 404.48,Z 231.591,A -85,B 0,C 180,E1 -10978.008,E2 -10978.008} C_VEL
LIN {X 0,Y 404.609,Z 231.56,A -85,B 0,C 180,E1 -10979.999,E2 -10979.999} C_VEL
LIN {X 0,Y 404.42,Z 231.604,A -85,B 0,C 180,E1 -10982.988,E2 -10982.988} C_VEL
LIN {X 0,Y 404.398,Z 231.605,A -85,B 0,C 180,E1 -10986.987,E2 -10986.987} C_VEL
LIN {X 0,Y 404.257,Z 231.603,A -85,B 0,C 180,E1 -10990.011,E2 -10990.011} C_VEL
LIN {X 0,Y 404.265,Z 231.624,A -85,B 0,C 180,E1 -10993.211,E2 -10993.211} C_VEL
LIN {X 0,Y 404.214,Z 231.624,A -85,B 0,C 180,E1 -10997.007,E2 -10997.007} C_VEL
LIN {X 0,Y 404.161,Z 231.625,A -85,B 0,C 180,E1 -11000.351,E2 -11000.351} C_VEL
LIN {X 0,Y 404.16,Z 231.639,A -85,B 0,C 180,E1 -11003.574,E2 -11003.574} C_VEL
LIN {X 0,Y 404.18,Z 231.633,A -85,B 0,C 180,E1 -11005.766,E2 -11005.766} C_VEL
LIN {X 0,Y 404.192,Z 231.619,A -85,B 0,C 180,E1 -11007.999,E2 -11007.999} C_VEL
LIN {X 0,Y 404.136,Z 231.643,A -85,B 0,C 180,E1 -11011.558,E2 -11011.558} C_VEL
LIN {X 0,Y 404.182,Z 231.626,A -85,B 0,C 180,E1 -11015.016,E2 -11015.016} C_VEL
LIN {X 0,Y 404.156,Z 231.638,A -85,B 0,C 180,E1 -11018.756,E2 -11018.756} C_VEL
LIN {X 0,Y 404.184,Z 231.629,A -85,B 0,C 180,E1 -11021.61,E2 -11021.61} C_VEL
LIN {X 0,Y 404.189,Z 231.632,A -85,B 0,C 180,E1 -11024.529,E2 -11024.529} C_VEL
LIN {X 0,Y 404.141,Z 231.613,A -85,B 0,C 180,E1 -11027.296,E2 -11027.296} C_VEL
LIN {X 0,Y 404.165,Z 231.626,A -85,B 0,C 180,E1 -11029.955,E2 -11029.955} C_VEL
LIN {X 0,Y 404.137,Z 231.643,A -85,B 0,C 180,E1 -11033.124,E2 -11033.124} C_VEL
LIN {X 0,Y 404.141,Z 231.627,A -85,B 0,C 180,E1 -11036.188,E2 -11036.188} C_VEL
LIN {X 0,Y 404.142,Z 231.632,A -85,B 0,C 180,E1 -11039.715,E2 -11039.715} C_VEL
LIN {X 0,Y 404.192,Z 231.639,A -85,B 0,C 180,E1 -11043.123,E2 -11043.123} C_VEL
LIN {X 0,Y 404.174,Z 231.642,A -85,B 0,C 180,E1 -11045.334,E2 -11045.334} C_VEL
LIN {X 0,Y 404.135,Z 231.645,A -85,B 0,C 180,E1 -11048.581,E2 -11048.581} C_VEL
LIN {X 0,Y 404.207,Z 231.637,A -85,B 0,C 180,E1 -11051.762,E2 -11051.762} C_VEL
LIN {X 0,Y 404.203,Z 231.638,A -85,B 0,C 180,E1 -11054.882,E2 -11054.882} C_VEL
LIN {X 0,Y 404.253,Z 231.631,A -85,B 0,C 180,E1 -11057.958,E2 -11057.958} C_VEL
LIN {X 0,Y 404.43,Z 231.61,A -85,B 0,C 180,E1 -11062.1,E2 -11062.1} C_VEL
LIN {X 0,Y 404.421,Z 231.61,A -85,B 0,C 180,E1 -11064.015,E2 -11064.015} C_VEL
LIN {X 0,Y 404.48,Z 231.603,A -85,B 0,C 180,E1 -11068.009,E2 -11068.009} C_VEL
LIN {X 0,Y 404.608,Z 231.588,A -85,B 0,C 180,E1 -11070,E2 -11070} C_VEL
LIN {X 0,Y 404.42,Z 231.611,A -85,B 0,C 180,E1 -11072.988,E2 -11072.988} C_VEL
LIN {X 0,Y 404.409,Z 231.613,A -85,B 0,C 180,E1 -11076.987,E2 -11076.987} C_VEL
LIN {X 0,Y 404.255,Z 231.631,A -85,B 0,C 180,E1 -11080.012,E2 -11080.012} C_VEL
LIN {X 0,Y 404.262,Z 231.631,A -85,B 0,C 180,E1 -11083.211,E2 -11083.211} C_VEL
LIN {X 0,Y 404.212,Z 231.637,A -85,B 0,C 180,E1 -11087.007,E2 -11087.007} C_VEL
LIN {X 0,Y 404.16,Z 231.644,A -85,B 0,C 180,E1 -11090.352,E2 -11090.352} C_VEL
LIN {X 0,Y 404.132,Z 231.644,A -85,B 0,C 180,E1 -11091.916,E2 -11091.916} C_VEL
LIN {X 0,Y 403.49,Z 231.728,A -85,B 0,C 180,E1 -11092.748,E2 -11092.748} C_VEL
LIN {X 0,Y 400.658,Z 232.085,A -85,B 0,C 180,E1 -11094.1,E2 -11094.1} C_VEL
LIN {X 0,Y 398.248,Z 232.386,A -85,B 0,C 180,E1 -11095.192,E2 -11095.192} C_VEL
LIN {X 0,Y 397.214,Z 232.511,A -85,B 0,C 180,E1 -11096.036,E2 -11096.036} C_VEL
LIN {X 0,Y 397.131,Z 232.518,A -85,B 0,C 180,E1 -11096.322,E2 -11096.322} C_VEL
LIN {X 0,Y 397.118,Z 232.504,A -85,B 0,C 180,E1 -11098.544,E2 -11098.544} C_VEL
LIN {X 0,Y 397.075,Z 232.526,A -85,B 0,C 180,E1 -11102.072,E2 -11102.072} C_VEL
LIN {X 0,Y 397.116,Z 232.501,A -85,B 0,C 180,E1 -11105.504,E2 -11105.504} C_VEL
LIN {X 0,Y 397.133,Z 232.513,A -85,B 0,C 180,E1 -11108.863,E2 -11108.863} C_VEL
LIN {X 0,Y 397.08,Z 232.488,A -85,B 0,C 180,E1 -11112.265,E2 -11112.265} C_VEL
LIN {X 0,Y 397.114,Z 232.512,A -85,B 0,C 180,E1 -11115.065,E2 -11115.065} C_VEL
LIN {X 0,Y 397.153,Z 232.509,A -85,B 0,C 180,E1 -11118.007,E2 -11118.007} C_VEL
LIN {X 0,Y 397.106,Z 232.52,A -85,B 0,C 180,E1 -11121.726,E2 -11121.726} C_VEL
LIN {X 0,Y 397.123,Z 232.504,A -85,B 0,C 180,E1 -11125.507,E2 -11125.507} C_VEL
LIN {X 0,Y 397.075,Z 232.522,A -85,B 0,C 180,E1 -11129.118,E2 -11129.118} C_VEL
LIN {X 0,Y 397.191,Z 232.487,A -85,B 0,C 180,E1 -11132.61,E2 -11132.61} C_VEL
LIN {X 0,Y 397.126,Z 232.518,A -85,B 0,C 180,E1 -11135.982,E2 -11135.982} C_VEL
LIN {X 0,Y 397.136,Z 232.498,A -85,B 0,C 180,E1 -11139.705,E2 -11139.705} C_VEL
LIN {X 0,Y 397.18,Z 232.499,A -85,B 0,C 180,E1 -11142.845,E2 -11142.845} C_VEL
LIN {X 0,Y 397.225,Z 232.501,A -85,B 0,C 180,E1 -11146.68,E2 -11146.68} C_VEL
LIN {X 0,Y 397.217,Z 232.48,A -85,B 0,C 180,E1 -11149.81,E2 -11149.81} C_VEL
LIN {X 0,Y 397.348,Z 232.481,A -85,B 0,C 180,E1 -11152.888,E2 -11152.888} C_VEL
LIN {X 0,Y 397.252,Z 232.501,A -85,B 0,C 180,E1 -11154.926,E2 -11154.926} C_VEL
LIN {X 0,Y 397.45,Z 232.461,A -85,B 0,C 180,E1 -11157.974,E2 -11157.974} C_VEL
LIN {X 0,Y 397.578,Z 232.435,A -85,B 0,C 180,E1 -11160.001,E2 -11160.001} C_VEL
LIN {X 0,Y 397.375,Z 232.482,A -85,B 0,C 180,E1 -11163.042,E2 -11163.042} C_VEL
LIN {X 0,Y 397.345,Z 232.485,A -85,B 0,C 180,E1 -11166.092,E2 -11166.092} C_VEL
LIN {X 0,Y 397.235,Z 232.478,A -85,B 0,C 180,E1 -11169.163,E2 -11169.163} C_VEL
LIN {X 0,Y 397.219,Z 232.496,A -85,B 0,C 180,E1 -11172.259,E2 -11172.259} C_VEL
LIN {X 0,Y 397.179,Z 232.504,A -85,B 0,C 180,E1 -11175.393,E2 -11175.393} C_VEL
LIN {X 0,Y 397.158,Z 232.491,A -85,B 0,C 180,E1 -11178.574,E2 -11178.574} C_VEL
LIN {X 0,Y 397.096,Z 232.515,A -85,B 0,C 180,E1 -11181.819,E2 -11181.819} C_VEL
LIN {X 0,Y 397.153,Z 232.5,A -85,B 0,C 180,E1 -11185.513,E2 -11185.513} C_VEL
LIN {X 0,Y 397.123,Z 232.508,A -85,B 0,C 180,E1 -11188.544,E2 -11188.544} C_VEL
LIN {X 0,Y 397.078,Z 232.522,A -85,B 0,C 180,E1 -11192.072,E2 -11192.072} C_VEL
LIN {X 0,Y 397.1,Z 232.513,A -85,B 0,C 180,E1 -11195.5,E2 -11195.5} C_VEL
LIN {X 0,Y 397.127,Z 232.51,A -85,B 0,C 180,E1 -11198.861,E2 -11198.861} C_VEL
LIN {X 0,Y 397.07,Z 232.526,A -85,B 0,C 180,E1 -11202.268,E2 -11202.268} C_VEL
LIN {X 0,Y 397.089,Z 232.518,A -85,B 0,C 180,E1 -11205.069,E2 -11205.069} C_VEL
LIN {X 0,Y 397.068,Z 232.517,A -85,B 0,C 180,E1 -11208.022,E2 -11208.022} C_VEL
LIN {X 0,Y 397.133,Z 232.512,A -85,B 0,C 180,E1 -11211.139,E2 -11211.139} C_VEL
LIN {X 0,Y 397.121,Z 232.507,A -85,B 0,C 180,E1 -11214.497,E2 -11214.497} C_VEL
LIN {X 0,Y 397.08,Z 232.516,A -85,B 0,C 180,E1 -11217.929,E2 -11217.929} C_VEL
LIN {X 0,Y 397.172,Z 232.699,A -85,B 0,C 180,E1 -11220.014,E2 -11220.014} C_VEL
LIN {X 0,Y 399.283,Z 243.577,A -85,B 0,C 180,E1 -11223.331,E2 -11223.331} C_VEL
LIN {X 0,Y 399.742,Z 248.784,A -85,B 0,C 180,E1 -11224.764,E2 -11224.764} C_VEL
LIN {X 0,Y 398.72,Z 262.093,A -85,B 0,C 180,E1 -11228.275,E2 -11228.275} C_VEL
LIN {X 0,Y 398.263,Z 267.961,A -85,B 0,C 180,E1 -11229.843,E2 -11229.843} C_VEL
LIN {X 0,Y 399.04,Z 272.291,A -85,B 0,C 180,E1 -11230.02,E2 -11230.02} C_VEL
LIN {X 0,Y 403.521,Z 297.35,A -85,B 0,C 180,E1 -11230.711,E2 -11230.711} C_VEL
LIN {X 0,Y 402.573,Z 372.863,A -85,B 0,C 180,E1 -11232.08,E2 -11232.08} C_VEL
LIN {X 0,Y 402.218,Z 383.634,A -85,B 0,C 180,E1 -11232.392,E2 -11232.392} C_VEL
LIN {X 0,Y 401.731,Z 392.735,A -85,B 0,C 180,E1 -11232.764,E2 -11232.764} C_VEL
LIN {X 0,Y 401.083,Z 403.097,A -85,B 0,C 180,E1 -11233.326,E2 -11233.326} C_VEL
LIN {X 0,Y 400.49,Z 412.232,A -85,B 0,C 180,E1 -11233.955,E2 -11233.955} C_VEL
LIN {X 0,Y 399.74,Z 421.228,A -85,B 0,C 180,E1 -11234.709,E2 -11234.709} C_VEL
LIN {X 0,Y 399.148,Z 428.828,A -85,B 0,C 180,E1 -11235.469,E2 -11235.469} C_VEL
LIN {X 0,Y 398.416,Z 437.486,A -85,B 0,C 180,E1 -11236.501,E2 -11236.501} C_VEL
LIN {X 0,Y 397.852,Z 444.575,A -85,B 0,C 180,E1 -11237.503,E2 -11237.503} C_VEL
LIN {X 0,Y 397.279,Z 450.776,A -85,B 0,C 180,E1 -11238.521,E2 -11238.521} C_VEL
LIN {X 0,Y 396.794,Z 457.315,A -85,B 0,C 180,E1 -11239.798,E2 -11239.798} C_VEL
LIN {X 0,Y 396.422,Z 461.816,A -85,B 0,C 180,E1 -11240.819,E2 -11240.819} C_VEL
LIN {X 0,Y 396.063,Z 467.307,A -85,B 0,C 180,E1 -11242.352,E2 -11242.352} C_VEL
LIN {X 0,Y 395.863,Z 471.632,A -85,B 0,C 180,E1 -11243.885,E2 -11243.885} C_VEL
LIN {X 0,Y 395.843,Z 473.999,A -85,B 0,C 180,E1 -11244.907,E2 -11244.907} C_VEL
LIN {X 0,Y 395.776,Z 475.797,A -85,B 0,C 180,E1 -11245.927,E2 -11245.927} C_VEL
LIN {X 0,Y 395.763,Z 478.241,A -85,B 0,C 180,E1 -11247.965,E2 -11247.965} C_VEL
LIN {X 0,Y 395.792,Z 478.83,A -85,B 0,C 180,E1 -11248.983,E2 -11248.983} C_VEL
LIN {X 0,Y 395.792,Z 478.83,A -85,B 0,C 180,E1 -11251.017,E2 -11251.017} C_VEL
LIN {X 0,Y 395.763,Z 478.241,A -85,B 0,C 180,E1 -11252.035,E2 -11252.035} C_VEL
LIN {X 0,Y 395.776,Z 475.797,A -85,B 0,C 180,E1 -11254.073,E2 -11254.073} C_VEL
LIN {X 0,Y 395.843,Z 473.999,A -85,B 0,C 180,E1 -11255.093,E2 -11255.093} C_VEL
LIN {X 0,Y 395.92,Z 470.393,A -85,B 0,C 180,E1 -11256.625,E2 -11256.625} C_VEL
LIN {X 0,Y 396.179,Z 465.647,A -85,B 0,C 180,E1 -11258.159,E2 -11258.159} C_VEL
LIN {X 0,Y 396.608,Z 459.626,A -85,B 0,C 180,E1 -11259.691,E2 -11259.691} C_VEL
LIN {X 0,Y 397.035,Z 453.528,A -85,B 0,C 180,E1 -11260.97,E2 -11260.97} C_VEL
LIN {X 0,Y 397.56,Z 447.828,A -85,B 0,C 180,E1 -11261.988,E2 -11261.988} C_VEL
LIN {X 0,Y 398.27,Z 439.273,A -85,B 0,C 180,E1 -11263.262,E2 -11263.262} C_VEL
LIN {X 0,Y 398.955,Z 431.093,A -85,B 0,C 180,E1 -11264.278,E2 -11264.278} C_VEL
LIN {X 0,Y 399.613,Z 422.715,A -85,B 0,C 180,E1 -11265.152,E2 -11265.152} C_VEL
LIN {X 0,Y 400.33,Z 413.863,A -85,B 0,C 180,E1 -11265.921,E2 -11265.921} C_VEL
LIN {X 0,Y 401.019,Z 404.104,A -85,B 0,C 180,E1 -11266.612,E2 -11266.612} C_VEL
LIN {X 0,Y 401.662,Z 394.023,A -85,B 0,C 180,E1 -11267.173,E2 -11267.173} C_VEL
LIN {X 0,Y 402.187,Z 384.509,A -85,B 0,C 180,E1 -11267.576,E2 -11267.576} C_VEL
LIN {X 0,Y 402.555,Z 374.195,A -85,B 0,C 180,E1 -11267.888,E2 -11267.888} C_VEL
LIN {X 0,Y 403.53,Z 301.199,A -85,B 0,C 180,E1 -11269.217,E2 -11269.217} C_VEL
LIN {X 0,Y 403.367,Z 296.269,A -85,B 0,C 180,E1 -11269.316,E2 -11269.316} C_VEL
LIN {X 0,Y 398.304,Z 268.431,A -85,B 0,C 180,E1 -11270.109,E2 -11270.109} C_VEL
LIN {X 0,Y 398.252,Z 267.413,A -85,B 0,C 180,E1 -11270.263,E2 -11270.263} C_VEL
LIN {X 0,Y 399.364,Z 254.157,A -85,B 0,C 180,E1 -11273.876,E2 -11273.876} C_VEL
LIN {X 0,Y 399.868,Z 248.06,A -85,B 0,C 180,E1 -11275.506,E2 -11275.506} C_VEL
LIN {X 0,Y 398.7,Z 240.392,A -85,B 0,C 180,E1 -11277.688,E2 -11277.688} C_VEL
LIN {X 0,Y 397.167,Z 232.563,A -85,B 0,C 180,E1 -11280.054,E2 -11280.054} C_VEL
LIN {X 0,Y 397.121,Z 232.52,A -85,B 0,C 180,E1 -11283.718,E2 -11283.718} C_VEL
LIN {X 0,Y 397.096,Z 232.519,A -85,B 0,C 180,E1 -11287.209,E2 -11287.209} C_VEL
LIN {X 0,Y 397.103,Z 232.499,A -85,B 0,C 180,E1 -11290.445,E2 -11290.445} C_VEL
LIN {X 0,Y 397.103,Z 232.523,A -85,B 0,C 180,E1 -11293.648,E2 -11293.648} C_VEL
LIN {X 0,Y 397.104,Z 232.517,A -85,B 0,C 180,E1 -11296.521,E2 -11296.521} C_VEL
LIN {X 0,Y 397.114,Z 232.51,A -85,B 0,C 180,E1 -11300.422,E2 -11300.422} C_VEL
LIN {X 0,Y 397.099,Z 232.52,A -85,B 0,C 180,E1 -11303.005,E2 -11303.005} C_VEL
LIN {X 0,Y 397.112,Z 232.505,A -85,B 0,C 180,E1 -11306.726,E2 -11306.726} C_VEL
LIN {X 0,Y 397.125,Z 232.513,A -85,B 0,C 180,E1 -11310.295,E2 -11310.295} C_VEL
LIN {X 0,Y 397.195,Z 232.493,A -85,B 0,C 180,E1 -11312.609,E2 -11312.609} C_VEL
LIN {X 0,Y 397.129,Z 232.513,A -85,B 0,C 180,E1 -11315.981,E2 -11315.981} C_VEL
LIN {X 0,Y 397.139,Z 232.5,A -85,B 0,C 180,E1 -11319.704,E2 -11319.704} C_VEL
LIN {X 0,Y 397.182,Z 232.493,A -85,B 0,C 180,E1 -11322.844,E2 -11322.844} C_VEL
LIN {X 0,Y 397.229,Z 232.503,A -85,B 0,C 180,E1 -11326.702,E2 -11326.702} C_VEL
LIN {X 0,Y 397.216,Z 232.48,A -85,B 0,C 180,E1 -11329.808,E2 -11329.808} C_VEL
LIN {X 0,Y 397.318,Z 232.484,A -85,B 0,C 180,E1 -11332.887,E2 -11332.887} C_VEL
LIN {X 0,Y 397.247,Z 232.504,A -85,B 0,C 180,E1 -11334.925,E2 -11334.925} C_VEL
LIN {X 0,Y 397.449,Z 232.467,A -85,B 0,C 180,E1 -11337.973,E2 -11337.973} C_VEL
LIN {X 0,Y 397.578,Z 232.435,A -85,B 0,C 180,E1 -11339.999,E2 -11339.999} C_VEL
LIN {X 0,Y 397.379,Z 232.482,A -85,B 0,C 180,E1 -11343.041,E2 -11343.041} C_VEL
LIN {X 0,Y 397.343,Z 232.483,A -85,B 0,C 180,E1 -11346.578,E2 -11346.578} C_VEL
LIN {X 0,Y 397.251,Z 232.477,A -85,B 0,C 180,E1 -11349.161,E2 -11349.161} C_VEL
LIN {X 0,Y 397.218,Z 232.495,A -85,B 0,C 180,E1 -11352.258,E2 -11352.258} C_VEL
LIN {X 0,Y 397.178,Z 232.507,A -85,B 0,C 180,E1 -11355.391,E2 -11355.391} C_VEL
LIN {X 0,Y 397.16,Z 232.492,A -85,B 0,C 180,E1 -11358.573,E2 -11358.573} C_VEL
LIN {X 0,Y 397.093,Z 232.515,A -85,B 0,C 180,E1 -11361.818,E2 -11361.818} C_VEL
LIN {X 0,Y 397.149,Z 232.507,A -85,B 0,C 180,E1 -11365.512,E2 -11365.512} C_VEL
LIN {X 0,Y 397.119,Z 232.507,A -85,B 0,C 180,E1 -11368.543,E2 -11368.543} C_VEL
LIN {X 0,Y 397.076,Z 232.524,A -85,B 0,C 180,E1 -11372.071,E2 -11372.071} C_VEL
LIN {X 0,Y 397.117,Z 232.507,A -85,B 0,C 180,E1 -11375.503,E2 -11375.503} C_VEL
LIN {X 0,Y 397.13,Z 232.513,A -85,B 0,C 180,E1 -11378.862,E2 -11378.862} C_VEL
LIN {X 0,Y 397.155,Z 232.514,A -85,B 0,C 180,E1 -11382.255,E2 -11382.255} C_VEL
LIN {X 0,Y 397.108,Z 232.513,A -85,B 0,C 180,E1 -11385.065,E2 -11385.065} C_VEL
LIN {X 0,Y 397.082,Z 232.488,A -85,B 0,C 180,E1 -11388.018,E2 -11388.018} C_VEL
LIN {X 0,Y 397.133,Z 232.513,A -85,B 0,C 180,E1 -11391.137,E2 -11391.137} C_VEL
LIN {X 0,Y 397.116,Z 232.501,A -85,B 0,C 180,E1 -11394.496,E2 -11394.496} C_VEL
LIN {X 0,Y 397.075,Z 232.526,A -85,B 0,C 180,E1 -11397.928,E2 -11397.928} C_VEL
LIN {X 0,Y 397.118,Z 232.505,A -85,B 0,C 180,E1 -11401.456,E2 -11401.456} C_VEL
LIN {X 0,Y 397.149,Z 232.515,A -85,B 0,C 180,E1 -11404.487,E2 -11404.487} C_VEL
LIN {X 0,Y 397.105,Z 232.522,A -85,B 0,C 180,E1 -11407.086,E2 -11407.086} C_VEL
LIN {X 0,Y 397.145,Z 232.516,A -85,B 0,C 180,E1 -11410.353,E2 -11410.353} C_VEL
LIN {X 0,Y 397.163,Z 232.515,A -85,B 0,C 180,E1 -11413.553,E2 -11413.553} C_VEL
LIN {X 0,Y 397.225,Z 232.507,A -85,B 0,C 180,E1 -11416.703,E2 -11416.703} C_VEL
LIN {X 0,Y 397.215,Z 232.509,A -85,B 0,C 180,E1 -11419.809,E2 -11419.809} C_VEL
LIN {X 0,Y 397.361,Z 232.491,A -85,B 0,C 180,E1 -11422.888,E2 -11422.888} C_VEL
LIN {X 0,Y 397.253,Z 232.504,A -85,B 0,C 180,E1 -11424.925,E2 -11424.925} C_VEL
LIN {X 0,Y 397.46,Z 232.769,A -85,B 0,C 180,E1 -11428.227,E2 -11428.227} C_VEL
LIN {X 0,Y 397.65,Z 232.873,A -85,B 0,C 180,E1 -11430,E2 -11430} C_VEL
LIN {X 0,Y 397.378,Z 232.565,A -85,B 0,C 180,E1 -11433.041,E2 -11433.041} C_VEL
LIN {X 0,Y 397.361,Z 232.491,A -85,B 0,C 180,E1 -11437.112,E2 -11437.112} C_VEL
LIN {X 0,Y 397.215,Z 232.509,A -85,B 0,C 180,E1 -11440.191,E2 -11440.191} C_VEL
LIN {X 0,Y 397.223,Z 232.507,A -85,B 0,C 180,E1 -11443.321,E2 -11443.321} C_VEL
LIN {X 0,Y 397.178,Z 232.513,A -85,B 0,C 180,E1 -11447.155,E2 -11447.155} C_VEL
LIN {X 0,Y 397.099,Z 232.523,A -85,B 0,C 180,E1 -11450.73,E2 -11450.73} C_VEL
LIN {X 0,Y 397.129,Z 232.519,A -85,B 0,C 180,E1 -11454.018,E2 -11454.018} C_VEL
LIN {X 0,Y 397.131,Z 232.518,A -85,B 0,C 180,E1 -11456.322,E2 -11456.322} C_VEL
LIN {X 0,Y 396.46,Z 232.602,A -85,B 0,C 180,E1 -11457.169,E2 -11457.169} C_VEL
LIN {X 0,Y 393.586,Z 232.944,A -85,B 0,C 180,E1 -11458.544,E2 -11458.544} C_VEL
LIN {X 0,Y 391.148,Z 233.246,A -85,B 0,C 180,E1 -11459.656,E2 -11459.656} C_VEL
LIN {X 0,Y 390.096,Z 233.384,A -85,B 0,C 180,E1 -11460.516,E2 -11460.516} C_VEL
LIN {X 0,Y 390.008,Z 233.394,A -85,B 0,C 180,E1 -11460.807,E2 -11460.807} C_VEL
LIN {X 0,Y 390.064,Z 233.377,A -85,B 0,C 180,E1 -11464.025,E2 -11464.025} C_VEL
LIN {X 0,Y 390.043,Z 233.398,A -85,B 0,C 180,E1 -11467.552,E2 -11467.552} C_VEL
LIN {X 0,Y 390.073,Z 233.371,A -85,B 0,C 180,E1 -11470.825,E2 -11470.825} C_VEL
LIN {X 0,Y 390.059,Z 233.389,A -85,B 0,C 180,E1 -11474.643,E2 -11474.643} C_VEL
LIN {X 0,Y 390.118,Z 233.39,A -85,B 0,C 180,E1 -11477.613,E2 -11477.613} C_VEL
LIN {X 0,Y 390.091,Z 233.39,A -85,B 0,C 180,E1 -11480.909,E2 -11480.909} C_VEL
LIN {X 0,Y 390.082,Z 233.382,A -85,B 0,C 180,E1 -11484.794,E2 -11484.794} C_VEL
LIN {X 0,Y 390.021,Z 233.401,A -85,B 0,C 180,E1 -11488.496,E2 -11488.496} C_VEL
LIN {X 0,Y 390.114,Z 233.371,A -85,B 0,C 180,E1 -11492.071,E2 -11492.071} C_VEL
LIN {X 0,Y 390.074,Z 233.393,A -85,B 0,C 180,E1 -11495.52,E2 -11495.52} C_VEL
LIN {X 0,Y 390.085,Z 233.379,A -85,B 0,C 180,E1 -11499.53,E2 -11499.53} C_VEL
LIN {X 0,Y 390.136,Z 233.379,A -85,B 0,C 180,E1 -11503.249,E2 -11503.249} C_VEL
LIN {X 0,Y 390.193,Z 233.377,A -85,B 0,C 180,E1 -11506.562,E2 -11506.562} C_VEL
LIN {X 0,Y 390.204,Z 233.353,A -85,B 0,C 180,E1 -11510.672,E2 -11510.672} C_VEL
LIN {X 0,Y 390.323,Z 233.363,A -85,B 0,C 180,E1 -11513.799,E2 -11513.799} C_VEL
LIN {X 0,Y 390.419,Z 233.337,A -85,B 0,C 180,E1 -11517.937,E2 -11517.937} C_VEL
